	KeyTimer		: TIME := T#200ms;
	sLux_EN			: FLT_EVENT;
	chkLux_ST		: FLT_TIME := ( TTAP:=T#20S, INITEV:=FALSE );
	chkLux_ST_Analog: FLT_TIME := ( TTAP:=T#20S, INITEV:=FALSE );
	HourMinNow		: STRING;
	semaphore		: BOOL:=GRUN;
	OnFromKey		: BOOL;
	fTrigFun		: F_TRIG;
	rTrigFun		: R_TRIG;
	fTrigKey		: F_TRIG;
	ActionKeyState	: en_ActionKey;
	KeyCounter, x	: BYTE;
	CtrlKey			: BOOL;
	DimmingValForKey: INT; (* valore 0...100 del dimming di default del lux sotto key *)
	ModeToServer : BYTE;
	ForcedOn : BYTE;
	ForcedOff : BYTE;

END_VAR
(* Con l'ID si identifica il numero del lux sul campo quindi il suo valore può variare da 1 a LUXM_MAX (attualmente 1...900) *)
IF (KeyMode = BUTTON_NO) OR (KeyMode = BUTTON_NC) THEN (* se si usano dei pulsanti sui vari digital input...*)
	KeyCounter := 0;
	FOR x:=0 TO  KeyQty-1 DO
		IF CtrlKeyList[x] = 1 THEN
			KeyCounter := KeyCounter + 1;
		END_IF
	END_FOR
	IF (KeyCounter MOD 2) = 0 THEN
		CtrlKey := FALSE;
	ELSE
		DimmingValForKey := DimmingValForKeyList[0]; (* In caso di pulsanti si prende il valore della posizione 0 dell'array *)
		CtrlKey := TRUE;
	END_IF
ELSE (* altrimenti se uso l'interruttore ne posso usare solo 1 nella posizione 0 dell'array *)
	IF (DimmingValForKeyMax) THEN
		DimmingValForKey := 0;
		FOR x:=0 TO  KeyQty-1 DO
			IF (CtrlKeyList[x] = 1) AND (DimmingValForKeyList[x] > DimmingValForKey)
			THEN
				DimmingValForKey := DimmingValForKeyList[x];
			END_IF
		END_FOR
	ELSIF NOT(DimmingValForKeyMax) THEN
		DimmingValForKey :=1000;
		FOR x:=0 TO  KeyQty-1 DO
			IF (CtrlKeyList[x] = 1) AND (DimmingValForKeyList[x] < DimmingValForKey)
			THEN
				DimmingValForKey := DimmingValForKeyList[x];
			END_IF
		END_FOR
	END_IF
	CtrlKey := 0;
	FOR x:=0 TO  KeyQty-1 DO
			CtrlKey := CtrlKey OR CtrlKeyList[x];
	END_FOR

END_IF

CASE DimmingType OF (* set dell' AsiTypeOut per sapere se eseguire il set di un analog out o di un digital out *)
	NO_DIMMING:	(* if no dimming we are using a digital output *)
		LuxTypeOut := DIGITAL; (* Set digital out mode *)
	DIMMING:	(*  if dimming we are using analog output *)
		LuxTypeOut := ANALOG; (* Set analog out mode *)
END_CASE

(* Control logic *)
(* Restore mode and value	*)
IF RestoreKey THEN
	CTRL_MODE := CTRL_MODE_BackUp;
END_IF

CASE CTRL_MODE OF
	ManualeOff: (*  0 Manuale Off *)
		(* Se commutazione arrivata da key durante funzionamento in timer o cronografo *)
		IF  NOT(CtrlKey) AND (ActionKey > NormalMode) AND ( ActionKeyState = SwitchOFF)THEN
			ActionKeyState := NormalMode;
			CTRL_MODE := CTRL_MODE_BackUp;
		ELSE
			CASE DimmingType OF
				NO_DIMMING:	(* if no dimming we are using a digital output *)
					LuxDigitalOut := TRUE; (* Lux spento (digital) *)
				DIMMING:	(*  if dimming we are using analog and digital output *)
					DimmerCtrl(); (* In caso di switch off in manuale è sempre zero anche se arriva da key *)
			END_CASE
		END_IF
	ManualeOn: (*  1 Manuale On *)
		(* Se commutazione arrivata da key durante funzionamento in timer o cronografo *)
		IF  NOT(CtrlKey) AND (ActionKey > NormalMode) AND ( ActionKeyState = SwitchON) THEN
			ActionKeyState := NormalMode;
			CTRL_MODE := CTRL_MODE_BackUp;
		ELSE
			CASE DimmingType OF
				NO_DIMMING:	(* if no dimming we are using a digital output *)
					LuxDigitalOut := FALSE; (* Lux acceso (digital) *)
				DIMMING:	(*  if dimming we are using analog and digital output  *)
					IF ActionKeyState = SwitchON THEN
						DimmerCtrlKeyOn(); (* Se il manuale on è settato a causa di un key si impongono i dati del key stesso *)
					ELSE
						DimmerCtrl();
					END_IF
			END_CASE
		END_IF
	Cronografo: (*  2 Cronografo *)
		IF  (CtrlKey) AND (ActionKey > NormalMode) THEN
			CASE  ActionKey OF
				SwitchON: 	(* Corrisponde al manuale ON *)
					CTRL_MODE := ManualeOn;
					ActionKeyState := SwitchON;
					CASE DimmingType OF
						NO_DIMMING:	(* if no dimming we are using a digital output *)
							LuxDigitalOut := FALSE; (* Lux acceso (digital) *)
						DIMMING:	(*  if dimming we are using analog and digital output  *)
							DimmerCtrlKeyOn();
					END_CASE

				SwitchOFF:	(* Corrisponde al manuale OFF  *)
					CTRL_MODE := ManualeOff;
					ActionKeyState := SwitchOFF;
					CASE DimmingType OF
						NO_DIMMING:	(* if no dimming we are using a digital output  *)
							LuxDigitalOut := TRUE; (* Lux spento (digital)  *)
						DIMMING:	(*  if dimming we are using analog and digital output  *)
							DimmerCtrlKeyOff();
					END_CASE
			END_CASE
		ELSE
			CASE DimmingType OF
				NO_DIMMING:	(* if no dimming we are using a digital output  *)
					IF ValInCronoInLux = 1000 (* OR ( LuxElement[i].PressKeyVisuOn)  *)
						THEN
						LuxDigitalOut := FALSE; (* Lux acceso (digital)  *)
						ELSE IF ValInCronoInLux = 0 (* OR ( NOT LuxElement[i].PressKeyVisuOn)  *)
							THEN
							LuxDigitalOut := TRUE; (* Lux spento (digital)  *)
						END_IF
					END_IF
				DIMMING:	(*  if dimming we are using analog output  *)
					DimmerCtrl();
			END_CASE
		END_IF
	Timer: (*  3 Timer   *)
	IF  (CtrlKey) AND (ActionKey > NormalMode) THEN
		CASE  ActionKey OF
			SwitchON: 	(* Corrisponde al manuale ON  *)
				CTRL_MODE := ManualeOn;
				ActionKeyState := SwitchON;
				CASE DimmingType OF
					NO_DIMMING:	(* if no dimming we are using a digital output  *)
						LuxDigitalOut := FALSE; (* Lux acceso (digital)  *)
					DIMMING:	(*  if dimming we are using analog and digital output   *)
						DimmerCtrlKeyOn();
				END_CASE

			SwitchOFF:	(* Corrisponde al manuale OFF  *)
				CTRL_MODE := ManualeOff;
				ActionKeyState := SwitchOFF;
				CASE DimmingType OF
					NO_DIMMING:	(* if no dimming we are using a digital output  *)
						LuxDigitalOut := TRUE; (* Lux spento (digital)  *)
					DIMMING:	(*  if dimming we are using analog and digital output  *)
						DimmerCtrlKeyOff();
				END_CASE
		END_CASE
	ELSE
		CASE DimmingType OF
			NO_DIMMING:	(* if no dimming we are using a digital output  *)
				HourMinNow:=CONCAT('TOD#', BYTE_TO_STRING(Sys.Time_Hour));
				HourMinNow:=CONCAT(HourMinNow, ':');
				HourMinNow:=CONCAT(HourMinNow, BYTE_TO_STRING(Sys.Time_Min));
				HourMinNow:=CONCAT(HourMinNow,':00');

				(* Trig timer *)
				TrigTimer.PT:=LuxTimer;
				TrigTimer(IN:= CtrlTrig);

				IF (((STRING_TO_TOD(HourMinNow) > HourMinStartOn) AND (STRING_TO_TOD(HourMinNow) < HourMinEndOn))  (* Se siamo nell'orario corretto  *)
				OR ((LuxDigitalOut = FALSE) AND (TrigTimer.Q = FALSE))) (* oppure si era acceso e adesso siamo passati fuori orario e dobbiamo spegnere  *)
				THEN
					IF TrigTimer.Q THEN
						LuxDigitalOut := FALSE; (* Lux acceso (digital)  *)
						ELSE
							LuxDigitalOut:= TRUE; (* Lux spento (digital)  *)
					END_IF
				END_IF
			DIMMING:	(*  if dimming we are using analog output  *)

				HourMinNow:=CONCAT('TOD#', BYTE_TO_STRING(Sys.Time_Hour));
				HourMinNow:=CONCAT(HourMinNow, ':');
				HourMinNow:=CONCAT(HourMinNow, BYTE_TO_STRING(Sys.Time_Min));
				HourMinNow:=CONCAT(HourMinNow,':00');

				(* Trig timer *)
				TrigTimer.PT:=LuxTimer;
				TrigTimer(IN:= CtrlTrig);

				IF (((STRING_TO_TOD(HourMinNow) > HourMinStartOn) AND (STRING_TO_TOD(HourMinNow) < HourMinEndOn))  (* Se siamo nell'orario corretto  *)
				OR ((LuxDigitalOut = FALSE) AND (TrigTimer.Q = FALSE))) (* oppure si era acceso e adesso siamo passati fuori orario e dobbiamo spegnere  *)
				THEN
					IF TrigTimer.Q THEN
						DimmerCtrl(); (* Lux acceso  *)
						ELSE
							LuxAnalogOut := 0; (* Lux spento  *)
							LuxDigitalOut := TRUE; (* Lux spento (digital)  *)
					END_IF
				END_IF
		END_CASE
		END_IF
	KeyControl: (*  4 Key function  *)
		IF CtrlKey THEN
			CASE DimmingType OF
				NO_DIMMING:	(* if no dimming we are using a digital output  *)
					LuxDigitalOut := FALSE; (* Lux acceso (digital)  *)
				DIMMING:	(*  if dimming we are using analog and digital output   *)
					DimmerCtrlKeyOn();
			END_CASE
		ELSIF CtrlKey = 0 THEN
			CASE DimmingType OF
				NO_DIMMING:	(* if no dimming we are using a digital output  *)
					LuxDigitalOut := TRUE; (* Lux spento (digital)  *)
				DIMMING:	(*  if dimming we are using analog and digital output  *)
					DimmerCtrlKeyOff();
			END_CASE
		END_IF
	END_CASE

(* ----------------------------------------------------------------------------------------------------------------------------------------  *)
(* Se i pin del feedback relè non sono cavallottati si usa la seguente riga al posto di quelle successive indicate da(#)  *)
(* REL_ST := LUX_ST[ID];	  																					 *)
(* ----------------------------------------------------------------------------------------------------------------------------------------   *)

(* setting della variabile REL_EN per compatibilità con il sw preesistente  *)
CASE DimmingType OF
	NO_DIMMING:	(* if no dimming we are using a digital output  *)
	IF LuxDigitalOut = TRUE  (* Lux spento  *)
		THEN
			(* Lux_State := FALSE;	//A causa del cavallotto sui pin del relè forzo a falso (#)  *)
			(* Lux_State := LUX_ST[ID];	  *)
			Lux_Enable := FALSE;
		ELSIF LuxDigitalOut = FALSE  (* Lux acceso			   *)
			THEN
				(* Lux_State := LUX_ST[ID];	//Quando so che la luce è accesa leggo lo stato del pin (che essendo cavallottato sarà a 1) (#)  *)
				Lux_Enable := TRUE;
	END_IF

	DIMMING:	(*  if dimming we are using analog output  *)
	IF LuxAnalogOut  = 0 (* Lux spento				  *)
		THEN
			(* REL_ST := FALSE;	 A causa del cavallotto sui pin del relè forzo a falso (#)  *)
			(* Lux_State := LUX_ST[ID];	  *)
			Lux_State:= TRUE;	(* aggiunta perchè non ho feedback sul relè *)
			Lux_Enable := FALSE;
			Lux_EnableAnalog := LuxAnalogOut; (* GIURE ver 008   *)
		ELSIF LuxAnalogOut > 0  (* Lux acceso			  *)
			THEN
				(* Lux_State := LUX_ST[ID];	 Quando so che la luce è accesa leggo lo stato del pin (che essendo cavallottato sarà a 1) (#)  *)
				Lux_State:= TRUE; (* aggiunta perchè non ho feedback sul relè *)
				Lux_Enable := TRUE;
				Lux_EnableAnalog := LuxAnalogOut;  (* GIURE ver 008  *)
	END_IF

END_CASE
(* Temporary energy counter *)
TickTimer(IN:=NOT TickTimer.Q);
IF TickTimer.Q AND Lux_Enable THEN
	LocalWorkingTime:=LocalWorkingTime+1;
	IF LocalEnergyCounter_t>36000000 THEN
		LocalEnergyCounter_t:=LocalEnergyCounter_t-36000000;
		LocalEnergyCounter:=LocalEnergyCounter+1;
	END_IF
END_IF

(* Generate status events *)
sLux_EN(IN:=Lux_Enable);
IF sLux_EN.EVL THEN
	LogEv(EL_Log,EO_LUX,ID,2,'Light OFF'); (* Light OFF  *)
END_IF
IF sLux_EN.EVH THEN
	LogEv(EL_Log,EO_LUX,ID,3,'Light ON'); (* Light ON  *)
	LocalPowerOnCycles:=LocalPowerOnCycles+1;
END_IF


(* Check status feedback *) (* GIURE ver 008 - aggiunta controllo valori analogici  *)
chkLux_ST_Analog(IN:=(Lux_StateAnalog<>Lux_EnableAnalog));
IF chkLux_ST_Analog.EVH THEN
	LogEv(EL_Alarm,EO_LUX,ID,9,'Fail Analog');(*  Feedback failure - Lux_StateAnalog<>Lux_EnableAnalog*)
END_IF
IF chkLux_ST_Analog.EVL THEN
	LogEv(EL_Log,EO_LUX,ID,1,'Successful Analog'); (*  Light feedback OK - Lux_StateAnalog = Lux_EnableAnalog  *)
END_IF
(* Check status feedback *)
chkLux_ST(IN:=(Lux_State<>Lux_Enable));
IF chkLux_ST.EVH THEN
	LogEv(EL_Alarm,EO_LUX,ID,9,'Fail'); (*  Feedback failure - Lux_State<>Lux_Enable  *)
END_IF
IF chkLux_ST.EVL THEN
	LogEv(EL_Log,EO_LUX,ID,1,'Successful'); (*  Light feedback OK - Lux_State = Lux_Enable  *)
END_IF


(* Status color *)
IF chkLux_ST.OUT THEN
	Status_Log:=2; Status_Vis:=COLOR_RED;
ELSE
	Status_Log:=0;
	Status_Vis:=SEL(Lux_Enable,COLOR_GREEN_OFF,COLOR_GREEN);
END_IF

(* Salvataggio dati in array ordinato per numero di ID utile per la visualizzazione  *)
DataLuxForVis[ID].VisStatus:=Status_Vis;
DataLuxForVis[ID].VisTimer:=LuxTimer/1000;
DataLuxForVis[ID].VisMod:=CTRL_MODE;
(* DataLuxForVis[ID].VisMod:=any_num_to_byte(CTRL_MODE); *)
END_FUNCTION_BLOCK
ACTION AddLogData:
Logger.s1:=INSERT('&LUX=',WORD_TO_STRING(ID),4);
IF ID<10 THEN Logger.s1:=INSERT(Logger.s1,'0',4); END_IF

Logger.s1:=CONCAT(Logger.s1,BOOL_TO_STRING(Lux_Enable));				Logger.s1:=CONCAT(Logger.s1,';');
Logger.s1:=CONCAT(Logger.s1,DWORD_TO_STRING(LocalWorkingTime));		Logger.s1:=CONCAT(Logger.s1,';');
Logger.s1:=CONCAT(Logger.s1,DWORD_TO_STRING(LocalPowerOnCycles));	Logger.s1:=CONCAT(Logger.s1,';');

CASE CTRL_MODE OF		(* modifica GIURE 009 ver 1.3 *)
	0: 	(*  Manuale OFF *)
		ModeToServer := 0;
		ForcedOn := 0;
		ForcedOff := 1;
	1:	(*  Manuale ON *)
		ModeToServer := 1;
		ForcedOn := 1;
		ForcedOff := 0;
	2:	(*  Cronografo *)
		ModeToServer := 2;
		ForcedOn := 0;
		ForcedOff := 0;
	3: 	(* Timer *)
		ModeToServer := 3;
		ForcedOn := 0;
		ForcedOff := 0;
END_CASE
Logger.s1:=CONCAT(Logger.s1,BYTE_TO_STRING(ModeToServer));			Logger.s1:=CONCAT(Logger.s1,';');
Logger.s1:=CONCAT(Logger.s1,BYTE_TO_STRING(Status_Log));				Logger.s1:=CONCAT(Logger.s1,';');
Logger.s1:=CONCAT(Logger.s1,BYTE_TO_STRING(ForcedOn));				Logger.s1:=CONCAT(Logger.s1,';');
Logger.s1:=CONCAT(Logger.s1,BYTE_TO_STRING(ForcedOff));				Logger.s1:=CONCAT(Logger.s1,';');
Logger.s1:=CONCAT(Logger.s1,BYTE_TO_STRING(DimmingType));			Logger.s1:=CONCAT(Logger.s1,';');
Logger.s1:=CONCAT(Logger.s1,WORD_TO_STRING(Lux_EnableAnalog/100));

ADDSTRING(ADR(Logger.TData), ADR(Logger.s1), Logger.TLen);
END_ACTION
ACTION DimmerCtrl:
CASE CTRL_MODE OF
	0: (* Manuale Off *)
		LuxAnalogOut := 0; (* Lux spento *)
		LuxDigitalOut := TRUE; (* Lux spento (digital) *)
	1: (* Manuale On *)
		LuxAnalogOut := 10000; (* Lux acceso *)
		LuxDigitalOut := FALSE; (* Lux acceso (digital) *)
	2: (* Cronografo *)
		IF ValInCronoInLux > 0 THEN
			LuxDigitalOut := FALSE; (* Lux acceso (digital) *)
			ELSE
				LuxDigitalOut := TRUE; (* Lux spento (digital) *)
		END_IF
		LuxAnalogOut := INT_TO_WORD(ValInCronoInLux*10);
	3: (* Timer 		 *)
		IF DimmingValForTimer > 0 THEN
			LuxDigitalOut := FALSE; (* Lux acceso (digital) *)
			ELSE
				LuxDigitalOut := TRUE; (* Lux spento (digital) *)
		END_IF
		LuxAnalogOut := INT_TO_WORD(DimmingValForTimer*10);
	ELSE (* default *)
		LuxDigitalOut := FALSE; (* Lux acceso (digital) *)
		LuxAnalogOut := 10000;
END_CASE
END_ACTION
ACTION DimmerCtrlKeyOff:
LuxAnalogOut := 0; (*/Lux spento*)
LuxDigitalOut := TRUE; (*Lux spento (digital)*)
END_ACTION
ACTION DimmerCtrlKeyOn:
LuxAnalogOut := INT_TO_WORD(DimmingValForKey*10);
LuxDigitalOut := FALSE; (*Lux acceso (digital) *)
END_ACTION
ACTION StatReset:
(* Reset statistic counters *)
LocalWorkingTime:=0;
LocalPowerOnCycles:=0;
LocalEnergyCounter:=0;
END_ACTION

(* POU Plant_Objects/obj_TPV, ST *)
FUNCTION_BLOCK obj_TPV
(* === TEMPERATURE PROBE  ===
   v1.0[16/04/15] - Versioning
*)
VAR CONSTANT
	NormalEv		: BYTE := 0;
	ErrorEv			: BYTE := 1;
	WarningEv		: BYTE := 2;
END_VAR
VAR_INPUT
	(* Settings *)
	ID				: BYTE;
	TAP				: BYTE:=4;	   (* Consecutive checks filter *)
	INITEV			: BOOL:= TRUE; (* Generate init OK event *)
	IN_EMIN			: INT :=-2000; (* Low error limit *)
	IN_WMIN			: INT := -550; (* Low warning value *)
	IN_WMAX			: INT :=  900; (* High warning value *)
	IN_EMAX			: INT := 8500; (* High error limit *)
	ERR_MIN_SHORT	: BOOL:= TRUE; (* TRUE  ==> EMIN=Short        , EMAX=Disconnected
									  FALSE ==> EMIN=Disconnected , EMAX=Short 		 *)
	(* Physical input *)
	IN			: INT;
END_VAR
VAR_OUTPUT
	WRN			: BOOL;	(* Value in warning range *)
	ERR			: BOOL;	(* Value error *)
	HI			: INT;	(* Highest value - cleared by Stat_Reset() action *)
	AVG			: INT; 	(* Average value - updated by Mean() action, cleared by Mean_Reset() action *)
	LOW			: INT;	(* Lowest value  - cleared by Stat_Reset() action *)

	Status_Log	: WORD;
	Status_Vis	: DWORD;
END_VAR
VAR
	cnt			: BYTE;
	event		: BYTE := 0;	(* 0: monitoring a generic, 1: monitoring an error, 2: monitoring a warning *)
	asum		: DINT;
	acnt		: WORD;
END_VAR
(* Check probe value limits *)
IF IN<=IN_EMIN OR IN>=IN_EMAX THEN
	IF NOT ERR THEN
		IF event <> ErrorEv THEN
			cnt := 1;
			event := ErrorEv;
		ELSE
			cnt:=cnt+1;
		END_IF

		IF cnt>TAP THEN
			cnt:=0;
			ERR:=TRUE; WRN:=FALSE;
			IF ( ERR_MIN_SHORT=TRUE  AND IN<=IN_EMIN ) OR ( ERR_MIN_SHORT=FALSE AND IN>=IN_EMAX ) THEN
				LogEv(EL_Alarm,EO_TPV,ID,5,INT_TO_STRING(IN));
			ELSE
				LogEv(EL_Alarm,EO_TPV,ID,4,INT_TO_STRING(IN));
			END_IF
		END_IF
	END_IF
ELSIF IN<=IN_WMIN OR IN>=IN_WMAX THEN
	IF NOT WRN THEN
		IF event <> WarningEv THEN
			cnt := 1;
			event := WarningEv;
		ELSE
			cnt:=cnt+1;
		END_IF

		IF cnt>TAP THEN
			cnt:=0;
			ERR:=FALSE; WRN:=TRUE;
			LogEv(EL_Wrn,EO_TPV,ID,SEL(IN<=IN_WMIN,3,2),INT_TO_STRING(IN));
		END_IF
	END_IF
ELSE
	IF INITEV OR WRN OR ERR THEN
		IF event <> NormalEv THEN
			cnt := 1;
			event := NormalEv;
		ELSE
			cnt:=cnt+1;
		END_IF

		IF cnt>TAP THEN
			cnt:=0;
			INITEV:=FALSE; ERR:=FALSE; WRN:=FALSE;
			LogEv(EL_Log,EO_TPV,ID,1,'Probe_OK');
		END_IF
	END_IF
END_IF


(*
(* Average value *)
IF acnt>=500 THEN
	Mean();
	asum := asum - AVG;
	acnt := acnt - 1;
END_IF

asum := asum + IN;
acnt := acnt + 1;
*)

AVG := IN;



(* Statistics values *)
IF IN<LOW THEN LOW:=IN; END_IF
IF IN>HI  THEN HI :=IN; END_IF

Lamp.obj_Status := Status_Log;
Lamp.UpdateStatus();

(* Status Log *)
IF ERR THEN	Status_Log := 2; Status_Vis := COLOR_RED;
ELSIF WRN THEN Status_Log := 1;	Status_Vis := COLOR_YELLOW;
ELSE Status_Log := 0; Status_Vis := COLOR_GREEN;
END_IF
END_FUNCTION_BLOCK
ACTION AddLogData:
Logger.s1:=INSERT('&TPV=',BYTE_TO_STRING(ID),4);
IF ID<10 THEN Logger.s1:=INSERT(Logger.s1,'0',4); END_IF
(*
Mean();
*)
Logger.s1:=CONCAT(Logger.s1,INT_TO_STRING(AVG));		Logger.s1:=CONCAT(Logger.s1,';');

Logger.s1:=CONCAT(Logger.s1,WORD_TO_STRING(Status_Log));
ADDSTRING(ADR(Logger.TData), ADR(Logger.s1), Logger.TLen);
END_ACTION
ACTION Mean:
(*AVG := DINT_TO_INT(asum/acnt); *)


AVG := IN;
END_ACTION
ACTION Mean_Reset:
AVG:=IN;
asum:=IN;
acnt:=1;
END_ACTION
ACTION Stat_Reset:
HI:=IN;
LOW:=IN;
END_ACTION

(* POU Plant_Objects/obj_VRD_new, ST *)
FUNCTION_BLOCK obj_VRD_new
(* === VALVOLA RIPARTITORE ===
   v1.0[16/04/15] - Versioning
*)
VAR CONSTANT
	Chk_CntSecAlarm	: INT := 900;	(* 900s = 15 minutes -> Observation itme *)
END_VAR
VAR_INPUT
	(* Settings *)
	ID				: BYTE;
	(* Controls *)
	RUN  			: BOOL;					(* Control input *)
	ReducedRange	: BOOL := FALSE;		(* If true output value is among 2 and 10V, otherwise 0-10V *)

	(* Physical inputs *)
	TEMP 			: INT;		(* Input temperature from sensor *)
	STATUS 			: WORD;		(* Input position from valve *)

	InitOK			: BOOL;
	Alarm1			: BOOL;
	Alarm2			: BOOL;
	Warning			: BOOL;

	Ctrl_Init		: BOOL;
	Ctrl_SetPoint	: INT;
	Ctrl_SetPointNew: INT := 0;
	Delta_SetPoint	: INT;
	Ctrl_Err		: INT;			(* Current error *)
	Ctrl_Err0		: INT; 			(* Previous error *)
	Ctrl_Accel		: REAL;			(* Derivate of error *)
	Ctrl_AccelGate  : INT:=1;		(* Derivate gate *)
	Ctrl_AccelTmr	: WORD;
	Ctrl_SetPointGate: INT := 5;	(* Setpoint gate - 0.5°C *)
	Ctrl_ErrGate	: INT:=5;		(* Error gate *)
	Ctrl_Kp			: REAL:=2;(*1;*)		(* Proportional factor *)
	Ctrl_Kd			: REAL:=10;(*100;*)  	(* Derivative factor *)
	Ctrl_Out		: REAL;

	Chk_Err			: INT;
	Chk_ErrGate		: INT:=1000; 		(* Check error gate *)
	Chk_Cnt			: INT;
	Chk_CntAlarm	: INT:=240; 		(* Check error trigger 120s *)

	(* Status *)
	Log_AvgTemp		: AVERAGE_T;
	Status_Log		: BYTE;
	Status_Vis 		: DWORD;

	(* Feedback *)
	fFeedback		: BOOL;			(* TRUE: Feedback available, FALSE: Feedback not available *)

	OffsetBoost: INT;

END_VAR
VAR_IN_OUT
(*	CLIM		: typ_Clima;  *)
END_VAR
VAR_OUTPUT
	(* Physical outputs *)
	OUT			: WORD;
END_VAR
VAR
	Curve		: CHARCURVE;
	Curve_Err	: BYTE;

	aTemp		: ARRAY [1..20] OF INT;
	meanTemp	: INT;
	sum			: INT := 0;
	Tmr			: TON := (PT:=T#1s);
	index		: BYTE;
	i			: BYTE;
	fCtrl_Err	: BOOL;		(* TRUE: Ctrl_Err>0, FALSE: Ctrl_Err<0 *)

	TON_AllarmeOvertemperatura:TON;


END_VAR


VAR_INPUT RETAIN
	Local_VRD_TAlarm: INT;
END_VAR
(* Check initialization *)
(*IF NOT InitOK THEN Init(); END_IF*)

(* Check max temperature *)

TON_AllarmeOvertemperatura(IN:=TEMP>Local_VRD_TAlarm,PT:=t#20s);
IF TON_AllarmeOvertemperatura.Q THEN
	IF NOT Alarm1 THEN
		Alarm1:=TRUE;
		LogEv(EL_AlarmStop,EO_VRD,ID,3,'VRD_Overtemperature');
	END_IF
END_IF

IF (TEMP<Local_VRD_TAlarm-10) AND Alarm1  THEN
		Alarm1:=FALSE;
END_IF




(* Check climatic setup *)
IF NOT CLIM.InitOK THEN	DefaultClim(); END_IF;
(* Calculate Setpoint *)
Curve(	IN:= T_AMB,	N:= 5, P:= CLIM.Points,			(* Given the x value as input, the corresponding y value as output is returned, if it matches the crve designed by array of points *)
		OUT=> Ctrl_SetPointNew, ERR=> Curve_Err );

IF Curve_Err>0 OR Ctrl_SetPoint>Plant_VRD_TMax THEN
	Ctrl_SetPoint:=Plant_VRD_TDefault;
	IF NOT Warning THEN
		Warning:=TRUE;
		LogEv(EL_Wrn,EO_VRD,ID,2,'VRD_Climatic_Error');
	END_IF
ELSE
	Delta_SetPoint := ABS(Ctrl_SetPoint - Ctrl_SetPointNew);
	IF Delta_SetPoint>Ctrl_SetPointGate THEN Ctrl_SetPoint := Ctrl_SetPointNew; END_IF

	Warning:=FALSE;
END_IF

Ctrl_SetPoint:=Ctrl_SetPoint+OffsetBoost;


(* Execute control loop [T=500ms] *)
(* IF RUN AND (NOT Alarm1) THEN*)
IF RUN  THEN
	(* Calculate error *)
	Ctrl_Err:=Ctrl_SetPoint-TEMP;
	(* Init/restart operations *)
	IF NOT Ctrl_Init THEN
		Ctrl_Accel:=0;
		Ctrl_AccelTmr:=0;
		Ctrl_Err0:=Ctrl_Err;
		Ctrl_Out:=5000;
		Ctrl_Init:=TRUE;
	END_IF
	(* Calculate acceleration *)
	IF ABS(Ctrl_Err-Ctrl_Err0)>Ctrl_AccelGate OR Ctrl_AccelTmr>20 THEN
		Ctrl_Accel:=INT_TO_REAL(Ctrl_Err-Ctrl_Err0)/WORD_TO_REAL(1+Ctrl_AccelTmr);
		Ctrl_AccelTmr:=0;
		Ctrl_Err0:=Ctrl_Err;
	ELSE
		Ctrl_AccelTmr:=Ctrl_AccelTmr+1;
	END_IF

	(* Gate error *)
	IF ABS(Ctrl_Err)>Ctrl_ErrGate THEN
		(* Control loop *)
		Ctrl_Out:=Ctrl_Out+(Ctrl_Kp*Ctrl_Err)+(Ctrl_Kd*Ctrl_Accel);
	END_IF

	(* Limiter and Output *)
(*	Ctrl_Out:=LIMIT(0,Ctrl_Out,27000); *)
	Ctrl_Out:=LIMIT(0,Ctrl_Out,32000);

ELSE
	Ctrl_Init:=FALSE;
	Ctrl_Out:=0;
END_IF

OUT:=SEL(Alarm1,REAL_TO_WORD(Ctrl_Out),0);





(* If there is an hardware feedback (such as 0-10V, potentiometer, ...) check it otherwise try to rebuild it *)
IF fFeedback THEN CheckFeedback();
ELSE BuildFeedback();
END_IF

(* Status temp *)
(* Status color *)
   IF Alarm1 THEN Status_Log:=2; Status_Vis:=16#2020F0;
ELSIF Warning  OR Alarm2        THEN Status_Log:=1; Status_Vis:=16#20F0F0;
                       ELSE Status_Log:=0; Status_Vis:=SEL(RUN,16#006000,16#20F020);
END_IF
END_FUNCTION_BLOCK
ACTION AddLogData:
Logger.s1:=INSERT('&VRD=',BYTE_TO_STRING(ID),4);
IF ID<10 THEN Logger.s1:=INSERT(Logger.s1,'0',4); END_IF


Logger.s1:=CONCAT(Logger.s1,INT_TO_STRING(Ctrl_SetPoint));				Logger.s1:=CONCAT(Logger.s1,';');

(* gli passo la percentuale di comando che ricavo dalla divisone per 327 del comando fisico *)
Logger.s1:=CONCAT(Logger.s1,WORD_TO_STRING(OUT/327));						Logger.s1:=CONCAT(Logger.s1,';');


(* gli passo la percentuale di apertura che ricavo dalla divisone per 327 del comando fisico *)
IF fFeedback THEN Logger.s1:=CONCAT(Logger.s1,WORD_TO_STRING(STATUS/327));
ELSE Logger.s1:=CONCAT(Logger.s1,'0');	(* Bypass *)
END_IF

Logger.s1:=CONCAT(Logger.s1,';');

Logger.s1:=CONCAT(Logger.s1,WORD_TO_STRING(Status_Log));

Logger.s1:=CONCAT(Logger.s1,';');
Logger.s1:=CONCAT(Logger.s1,'1'); (* Valvola modulante controllata Analogica *)

ADDSTRING(ADR(Logger.TData), ADR(Logger.s1), Logger.TLen);
END_ACTION
ACTION BuildFeedback:
(* Comparison is taken between actual temperature vs windowed mean value of last 20 temperature
   (check is carried out every second)	*)
IF RUN AND (NOT Alarm1) THEN

	IF Ctrl_Err>0 THEN
		IF NOT fCtrl_Err THEN index := 0; END_IF
		fCtrl_Err := TRUE;
	ELSE
		IF fCtrl_Err THEN index := 0; END_IF
		fCtrl_Err := FALSE;
	END_IF

	(* Temperature is lower than setpoint -->> Should increase *)
	Tmr(IN:=NOT Tmr.Q);

	IF Tmr.Q THEN

		IF index<21 THEN
			(* Fullfil temperature array *)
			aTemp[index] := TEMP;
			index := index + 1;

			IF index=20 THEN
				FOR i:=1 TO 20 BY 1 DO sum := sum + aTemp[i]; END_FOR
			END_IF
		ELSE
			(* Calculate mean value *)
			meanTemp := sum/20;

			IF (fCtrl_Err AND TEMP<meanTemp) OR (NOT fCtrl_Err AND TEMP>meanTemp) THEN

				IF Chk_Cnt>Chk_CntSecAlarm THEN
					IF NOT Alarm2 THEN
						Alarm2:=TRUE;
						LogEv(EL_Alarm,EO_VRD,ID,4,'VRD_Position_Error');
					END_IF
				ELSE
					Chk_Cnt := Chk_Cnt+1;
				END_IF

			ELSE
				(* Reset counter and alarm flag *)
				Chk_Cnt:=0;
				Alarm2:=FALSE;
			END_IF

			sum := 0;	(* Reset sum counter *)

			(* Shift array removing oldest value *)
			FOR i:=1 TO 20 BY 1 DO
				aTemp[i-1] := aTemp[i];
				sum := sum + aTemp[i];
			END_FOR

			aTemp[20] := TEMP;			(* Last temperature value is new one *)
			sum := sum + aTemp[20];		(* Update sum *)
		END_IF
	END_IF
END_IF
END_ACTION
ACTION CheckFeedback:
(* Calculate position error according to feedback *)
IF ReducedRange THEN
(* SETPOINT[2..10V]-STATUS[0..10V] *)
	IF OUT<=6553 THEN Chk_Err:=0; ELSE Chk_Err:=(OUT-6553)/262; END_IF
	Chk_Err:=(Chk_Err-STATUS)/327;
ELSE
(* SETPOINT[0..10V]-STATUS[0..10V] *)
	Chk_Err := OUT - STATUS;
END_IF

(* Check position error *)
IF ( ABS(Chk_Err)>Chk_ErrGate ) THEN
	IF Chk_Cnt>Chk_CntAlarm THEN
		IF NOT Alarm2 THEN
			Alarm2:=TRUE;
			LogEv(EL_Wrn,EO_VRD,ID,4,'VRD_Position_Error');
		END_IF
	ELSE
		Chk_Cnt:=Chk_Cnt+1;
	END_IF
ELSE
	Chk_Cnt:=0;
	Alarm2:=FALSE;
END_IF
END_ACTION
ACTION DefaultClim:
(*CLIM.Points[0].X:=-300; CLIM.Points[0].Y:=400;
CLIM.Points[1].X:=-50;  CLIM.Points[1].Y:=400;
CLIM.Points[2].X:= 200; CLIM.Points[2].Y:=200;
CLIM.Points[3].X:= 300; CLIM.Points[3].Y:=200;
CLIM.Points[4].X:= 500; CLIM.Points[4].Y:=200;*)
CLIM.Points[0].X:=-300; CLIM.Points[0].Y:=850;
CLIM.Points[1].X:=-50;  CLIM.Points[1].Y:=650;
CLIM.Points[2].X:= 100; CLIM.Points[2].Y:=400;
CLIM.Points[3].X:= 200; CLIM.Points[3].Y:=200;
CLIM.Points[4].X:= 500; CLIM.Points[4].Y:=200;
CLIM.InitOK:=TRUE;
LogEv(EL_Wrn,EO_VRD,ID,1,'Climatic_Default');
END_ACTION
ACTION Init:
(* End initialization *)
InitOK:=TRUE;
END_ACTION

(* POU Utils Functions/PLANT_STATUS, ST *)
FUNCTION_BLOCK PLANT_STATUS
VAR_INPUT
	obj_Status		:	WORD;
END_VAR
VAR_OUTPUT
END_VAR
VAR
	PLANT_STATUS	:	WORD;

	Pwm				:	TON := (PT:=T#1s);
END_VAR
CASE plant_Status OF

	0:	(* Plant OK - Everything works well *)
		(*Pwm(IN:=FALSE);	*)						(* Stop timer if running *)
		LAMP_AL := FALSE;						(* Keep the lamp switched off *)

	(*1:	(* Plant in warning *)
		Pwm(IN:= NOT(Pwm.Q));

		IF Pwm.Q THEN
			LAMP_AL := NOT LAMP_AL;				(* Toggle output *)
		END_IF*)

	2:	(* Plant in alarm *)
		(*Pwm(IN:=FALSE);	*)						(* Stop timer if running *)
		LAMP_AL	:= TRUE;						(* Keep the lamp switched on *)

END_CASE

plant_Status := 0;		(* Reset plant status *)
END_FUNCTION_BLOCK
ACTION UpdateStatus:
IF plant_Status = 2 THEN

	RETURN;					(* If plant already in alarm condition do nothing *)

ELSE

		IF obj_Status <> 0 THEN
			plant_Status := obj_Status;			(* If plant in warning/normal condition and current object in alarm, update plant status *)
		END_IF
END_IF
END_ACTION

(* POU PLC_WDT, ST *)
FUNCTION PLC_WDT: DWORD VAR_INPUT dwEvent: DWORD; dwFilter: DWORD; dwOwner: DWORD; END_VAR
LogEv(EL_AlarmStop,EO_SYS,1,10,'Watchdog');
END_FUNCTION

(* POU Utils Functions/RAWTOHEXSTR, ST *)
FUNCTION RAWTOHEXSTR : STRING(128)
VAR_INPUT
	pData: POINTER TO BYTE;
	DataLen: BYTE;
END_VAR
VAR
	pt: POINTER TO BYTE;
	xl: BYTE;
END_VAR
pt:=ADR(RAWTOHEXSTR);

xl:=2;

WHILE DataLen>0 AND xl<128 DO

	pt^ := (pData^ / 16#10) + 48 + (((pData^ / 16#10)/10)*7);
	pt:=pt+1;
	pt^ := (pData^ AND 16#0F)  + 48 + (((pData^ AND 16#0F)/10)*7);
	pt:=pt+1;

	xl:=xl+2;

	DataLen:=DataLen-1;
	pData:=pData+1;

END_WHILE

pt^:=0;
END_FUNCTION

(* POU Utils/RTC_Update, ST *)
FUNCTION RTC_Update : BOOL
VAR
	T: DT;
	TS: STRING;
	TS2: STRING;
	Hour: BYTE;
	Minute: BYTE;
END_VAR
(* Get RTC time *)
T:=SysRtcGetTime(TRUE);
Sys.Time_CT_DT:=T;
(* Calculate variables *)
TS:=DT_TO_STRING(T);
Sys.Time_LogString:=DELETE(STR:=TS, LEN:=3, POS:=1);
TS2:=MID(STR:=TS, LEN:=4, POS:= 4); Sys.Time_Year 	:=STRING_TO_WORD(TS2);
TS2:=MID(STR:=TS, LEN:=2, POS:= 9); Sys.Time_Month	:=STRING_TO_BYTE(TS2);
TS2:=MID(STR:=TS, LEN:=2, POS:=12); Sys.Time_Day  	:=STRING_TO_BYTE(TS2);
Sys.Time_CT_Day:=(32*(Sys.Time_Month-1)+Sys.Time_Day-1);
TS2:=MID(STR:=TS, LEN:=2, POS:=15); Hour			:=STRING_TO_BYTE(TS2);
TS2:=MID(STR:=TS, LEN:=2, POS:=18); Minute		 	:=STRING_TO_BYTE(TS2);
Sys.Time_Hour := Hour;
Sys.Time_Minute := Minute;
Sys.Time_CT_Quarter:=Hour*4+(Minute/15);
Sys.Time_CT_Minute:=Hour*60+Minute;
END_FUNCTION

(* POU Utils Functions/SHIFT_ARRAY, ST *)
FUNCTION SHIFT_ARRAY : BOOL
VAR_INPUT
	pData	:	POINTER TO ARRAY [1..2] OF WORD;
	Size	:	BYTE;
END_VAR
VAR
	pNew	:	POINTER TO WORD;
	i		:	BYTE;
END_VAR
(* Shift right *)
FOR i:=1 TO (Size-1) BY 1 DO

	(*pNew := pData + 1;*)
	pData^[i] := pData^[i+1];
	(*pData := pData + 1;*)

END_FOR
END_FUNCTION

(* POU Utils Functions/TONOF, ST *)
FUNCTION_BLOCK TONOF
VAR_INPUT
	IN		: BOOL;
	PT_ON	: TIME; (* time to pass, before OUT is set *)
	PT_OF	: TIME; (* time to pass, before OUT is reset *)
END_VAR
VAR_OUTPUT
	OUT		: BOOL;
END_VAR
VAR
	timer	: TON;
END_VAR
IF IN<>OUT THEN
	timer(IN:=TRUE,PT:=SEL(IN,PT_OF,PT_ON));
	IF timer.Q THEN OUT:=IN; END_IF
ELSE
	timer(IN:=FALSE);
END_IF
END_FUNCTION_BLOCK

(* Visualisation PLC_VISU
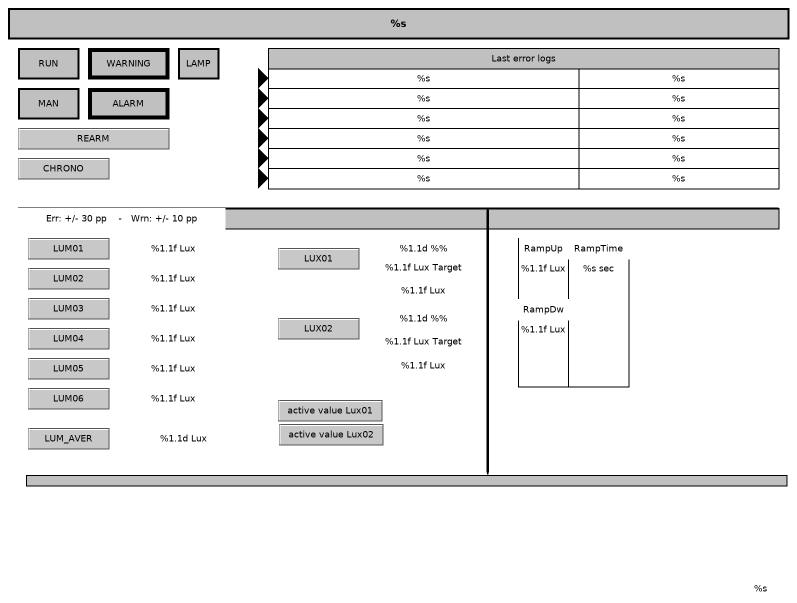
rectangle at (10,10)-(791,41): text "%s"; shows .Plant_NAME
rectangle at (530,580)-(771,601): text "%s"; shows Sys.Time_LogString
rounded rectangle at (20,50)-(81,81): text "RUN"; alarm colour if NOT Mode_Manual; runs INTERN ASSIGN Mode_Manual:=(FALSE)
rounded rectangle at (20,90)-(81,121): text "MAN"; alarm colour if Mode_Manual; runs INTERN ASSIGN Mode_Manual:=(TRUE)
rectangle at (580,70)-(781,91): text "%s"; shows Sys.LastLogs_Msg[0]
polygon at (260,170)-(270,190): invisible if Sys.LastLogs_Idx<>0
rectangle at (580,90)-(781,111): text "%s"; shows Sys.LastLogs_Msg[1]
polygon at (260,70)-(270,90): invisible if Sys.LastLogs_Idx<>1
rectangle at (580,110)-(781,131): text "%s"; shows Sys.LastLogs_Msg[2]
polygon at (260,90)-(270,110): invisible if Sys.LastLogs_Idx<>2
rectangle at (580,130)-(781,151): text "%s"; shows Sys.LastLogs_Msg[3]
polygon at (260,110)-(270,130): invisible if Sys.LastLogs_Idx<>3
rectangle at (580,150)-(781,171): text "%s"; shows Sys.LastLogs_Msg[4]
polygon at (260,130)-(270,150): invisible if Sys.LastLogs_Idx<>4
rectangle at (580,170)-(781,191): text "%s"; shows Sys.LastLogs_Msg[5]
polygon at (260,150)-(270,170): invisible if Sys.LastLogs_Idx<>5
rectangle at (270,70)-(581,91): text "%s"; shows Sys.LastLogs_Dat[0]
rectangle at (270,90)-(581,111): text "%s"; shows Sys.LastLogs_Dat[1]
rectangle at (270,110)-(581,131): text "%s"; shows Sys.LastLogs_Dat[2]
rectangle at (270,130)-(581,151): text "%s"; shows Sys.LastLogs_Dat[3]
rectangle at (270,150)-(581,171): text "%s"; shows Sys.LastLogs_Dat[4]
rectangle at (270,170)-(581,191): text "%s"; shows Sys.LastLogs_Dat[5]
rectangle at (90,90)-(171,121): text "ALARM"; alarm colour if Sys.Alarm; runs INTERN ASSIGN Mode_Manual:=(FALSE)
rectangle at (90,50)-(171,81): text "WARNING"; alarm colour if Sys.Warning; runs INTERN ASSIGN Mode_Manual:=(TRUE)
button at (20,130)-(171,151): text "REARM"; runs INTERN ASSIGN Sys.Alarm:=(FALSE);INTERN ASSIGN Sys.Warning:=(FALSE)
rectangle at (270,50)-(781,71): text "Last error logs"
rectangle at (520,240)-(571,261): text "RampUp"
rectangle at (520,260)-(571,281): text "%1.1f Lux"; shows RampUp*LuxSuBit
rounded rectangle at (180,50)-(221,81): text "LAMP"; alarm colour if LAMP_AL
button at (20,160)-(111,181): text "CHRONO"; opens VIS_CHONOEDITOR
button at (30,240)-(111,261): text "LUM01"
rectangle at (130,240)-(221,261): text "%1.1f Lux"; shows INT_TO_REAL(LumList[1].IN)*LuxSuBit
button at (30,270)-(111,291): text "LUM02"
rectangle at (130,270)-(221,291): text "%1.1f Lux"; shows INT_TO_REAL(LumList[2].IN)*LuxSuBit
button at (30,300)-(111,321): text "LUM03"
rectangle at (130,300)-(221,321): text "%1.1f Lux"; shows INT_TO_REAL(LumList[3].IN)*LuxSuBit
button at (30,330)-(111,351): text "LUM04"
rectangle at (130,330)-(221,351): text "%1.1f Lux"; shows INT_TO_REAL(LumList[4].IN)*LuxSuBit
button at (30,360)-(111,381): text "LUM05"
rectangle at (130,360)-(221,381): text "%1.1f Lux"; shows INT_TO_REAL(LumList[5].IN)*LuxSuBit
button at (30,390)-(111,411): text "LUM06"
rectangle at (130,390)-(221,411): text "%1.1f Lux"; shows DWORD_TO_REAL(LumList[6].IN)*LuxSuBit
button at (30,430)-(111,451): text "LUM_AVER"
rectangle at (140,430)-(231,451): text "%1.1d Lux"; shows PLC_PRG.LumValueAverageLux
button at (280,250)-(361,271): text "LUX01"
rectangle at (380,240)-(471,261): text "%1.1d %%"; shows LuxOutput[1].AnalogOut/100
rectangle at (380,282)-(471,303): text "%1.1f Lux"; shows INT_TO_REAL(LUX01)*LuxSuBit
button at (280,320)-(361,341): text "LUX02"
rectangle at (380,310)-(471,331): text "%1.1d %%"; shows LuxOutput[2].AnalogOut/100
rectangle at (380,357)-(471,378): text "%1.1f Lux"; shows INT_TO_REAL(LUX02)*LuxSuBit
rectangle at (520,301)-(571,322): text "RampDw"
rectangle at (520,321)-(571,342): text "%1.1f Lux"; shows RampDown*LuxSuBit
rectangle at (570,240)-(631,261): text "RampTime"
rectangle at (570,260)-(631,281): text "%s sec"; shows RampTime
rectangle at (20,210)-(227,231): text "Err: +/- 30 pp    -   Wrn: +/- 10 pp"
button at (280,402)-(384,423): text "active value Lux01"; toggles PLC_PRG.ValInCronoFromVisu[1]
button at (281,426)-(385,447): text "active value Lux02"; toggles PLC_PRG.ValInCronoFromVisu[2]
rectangle at (380,333)-(471,354): text "%1.1f Lux Target"; shows LuxOutput[2].AnalogOut*3.27*LuxSuBit
rectangle at (380,259)-(471,280): text "%1.1f Lux Target"; shows LuxOutput[1].AnalogOut*3.27*LuxSuBit
7 more shapes without text or variables
10 elements of other kinds (tables, trends, ...) not read
*)

(* Visualisation VIS_CHONOEDITOR
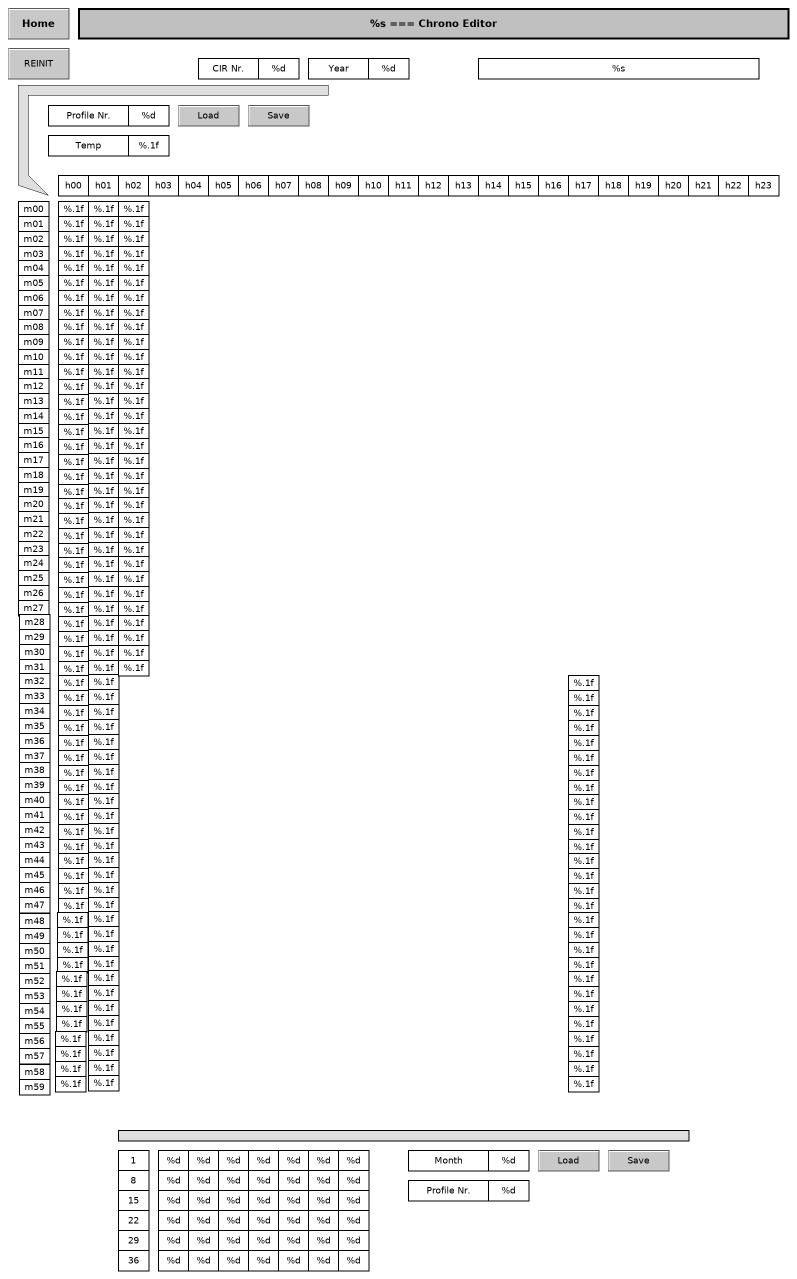
rectangle at (200,60)-(261,81): text "CIR Nr."
rectangle at (260,60)-(301,81): text "%d"; shows CronEd.CN_Sel; alarm colour if CronEd.CN_Sel<>CronEd.CN_Act; editable 1..250
rectangle at (50,107)-(131,128): text "Profile Nr."
rectangle at (130,107)-(171,128): text "%d"; shows CronEd.PR_Sel; alarm colour if CronEd.PR_Sel<>CronEd.PR_Act; editable 1..10
rectangle at (50,137)-(131,158): text "Temp"
rectangle at (130,137)-(171,158): text "%.1f"; shows CronEd.PR_TT; editable
button at (180,107)-(241,128): text "Load"; toggles CronEd.PR_Load
button at (250,107)-(311,128): text "Save"; toggles CronEd.PR_Save
rectangle at (20,203)-(51,219): text "m00"
rectangle at (20,218)-(51,234): text "m01"
rectangle at (20,233)-(51,249): text "m02"
rectangle at (20,248)-(51,264): text "m03"
rectangle at (80,10)-(791,41): text "%s === Chrono Editor"; shows .Plant_NAME
button at (10,10)-(71,41): text "Home"; opens PLC_VISU
rounded rectangle at (60,203)-(91,219): text "%.1f"; shows WORD_TO_REAL(CronEd.PR.Setpoint[0])/10; runs INTERN ASSIGN CronEd.PR.Setpoint[0]:=(REAL_TO_WORD(CronEd.PR_TT*10))
rounded rectangle at (60,218)-(91,234): text "%.1f"; shows WORD_TO_REAL(CronEd.PR.Setpoint[1])/10; runs INTERN ASSIGN CronEd.PR.Setpoint[1]:=(REAL_TO_WORD(CronEd.PR_TT*10))
rounded rectangle at (60,233)-(91,249): text "%.1f"; shows WORD_TO_REAL(CronEd.PR.Setpoint[2])/10; runs INTERN ASSIGN CronEd.PR.Setpoint[2]:=(REAL_TO_WORD(CronEd.PR_TT*10))
rounded rectangle at (60,248)-(91,264): text "%.1f"; shows WORD_TO_REAL(CronEd.PR.Setpoint[3])/10; runs INTERN ASSIGN CronEd.PR.Setpoint[3]:=(REAL_TO_WORD(CronEd.PR_TT*10))
rectangle at (60,177)-(91,198): text "h00"; runs INTERN ASSIGN CronEd.PR.Setpoint[0]:=(REAL_TO_WORD(CronEd.PR_TT*10));INTERN ASSIGN CronEd.PR.Setpoint[1]:=(REAL_TO_WORD(CronEd.PR_TT*10));INTERN ASSIGN CronEd.PR.Setpoint[2]:=(REAL_TO_WORD(CronEd.PR_TT*10));INTERN ASSIGN CronEd.PR.Setpoint[3]:=(REAL_TO_WORD(CronEd.PR_TT*10))
rectangle at (90,177)-(121,198): text "h01"; runs INTERN ASSIGN CronEd.PR.Setpoint[4]:=(REAL_TO_WORD(CronEd.PR_TT*10));INTERN ASSIGN CronEd.PR.Setpoint[5]:=(REAL_TO_WORD(CronEd.PR_TT*10));INTERN ASSIGN CronEd.PR.Setpoint[6]:=(REAL_TO_WORD(CronEd.PR_TT*10));INTERN ASSIGN CronEd.PR.Setpoint[7]:=(REAL_TO_WORD(CronEd.PR_TT*10))
rectangle at (120,177)-(151,198): text "h02"; runs INTERN ASSIGN CronEd.PR.Setpoint[8]:=(REAL_TO_WORD(CronEd.PR_TT*10));INTERN ASSIGN CronEd.PR.Setpoint[9]:=(REAL_TO_WORD(CronEd.PR_TT*10));INTERN ASSIGN CronEd.PR.Setpoint[10]:=(REAL_TO_WORD(CronEd.PR_TT*10));INTERN ASSIGN CronEd.PR.Setpoint[11]:=(REAL_TO_WORD(CronEd.PR_TT*10))
rectangle at (150,177)-(181,198): text "h03"; runs INTERN ASSIGN CronEd.PR.Setpoint[15]:=(REAL_TO_WORD(CronEd.PR_TT*10));INTERN ASSIGN CronEd.PR.Setpoint[14]:=(REAL_TO_WORD(CronEd.PR_TT*10));INTERN ASSIGN CronEd.PR.Setpoint[13]:=(REAL_TO_WORD(CronEd.PR_TT*10));INTERN ASSIGN CronEd.PR.Setpoint[12]:=(REAL_TO_WORD(CronEd.PR_TT*10))
rectangle at (180,177)-(211,198): text "h04"; runs INTERN ASSIGN CronEd.PR.Setpoint[19]:=(REAL_TO_WORD(CronEd.PR_TT*10));INTERN ASSIGN CronEd.PR.Setpoint[18]:=(REAL_TO_WORD(CronEd.PR_TT*10));INTERN ASSIGN CronEd.PR.Setpoint[17]:=(REAL_TO_WORD(CronEd.PR_TT*10));INTERN ASSIGN CronEd.PR.Setpoint[16]:=(REAL_TO_WORD(CronEd.PR_TT*10))
rectangle at (210,177)-(241,198): text "h05"; runs INTERN ASSIGN CronEd.PR.Setpoint[23]:=(REAL_TO_WORD(CronEd.PR_TT*10));INTERN ASSIGN CronEd.PR.Setpoint[22]:=(REAL_TO_WORD(CronEd.PR_TT*10));INTERN ASSIGN CronEd.PR.Setpoint[21]:=(REAL_TO_WORD(CronEd.PR_TT*10));INTERN ASSIGN CronEd.PR.Setpoint[20]:=(REAL_TO_WORD(CronEd.PR_TT*10))
rectangle at (240,177)-(271,198): text "h06"; runs INTERN ASSIGN CronEd.PR.Setpoint[27]:=(REAL_TO_WORD(CronEd.PR_TT*10));INTERN ASSIGN CronEd.PR.Setpoint[26]:=(REAL_TO_WORD(CronEd.PR_TT*10));INTERN ASSIGN CronEd.PR.Setpoint[25]:=(REAL_TO_WORD(CronEd.PR_TT*10));INTERN ASSIGN CronEd.PR.Setpoint[24]:=(REAL_TO_WORD(CronEd.PR_TT*10))
rectangle at (270,177)-(301,198): text "h07"; runs INTERN ASSIGN CronEd.PR.Setpoint[31]:=(REAL_TO_WORD(CronEd.PR_TT*10));INTERN ASSIGN CronEd.PR.Setpoint[30]:=(REAL_TO_WORD(CronEd.PR_TT*10));INTERN ASSIGN CronEd.PR.Setpoint[29]:=(REAL_TO_WORD(CronEd.PR_TT*10));INTERN ASSIGN CronEd.PR.Setpoint[28]:=(REAL_TO_WORD(CronEd.PR_TT*10))
rectangle at (300,177)-(331,198): text "h08"; runs INTERN ASSIGN CronEd.PR.Setpoint[35]:=(REAL_TO_WORD(CronEd.PR_TT*10));INTERN ASSIGN CronEd.PR.Setpoint[34]:=(REAL_TO_WORD(CronEd.PR_TT*10));INTERN ASSIGN CronEd.PR.Setpoint[33]:=(REAL_TO_WORD(CronEd.PR_TT*10));INTERN ASSIGN CronEd.PR.Setpoint[32]:=(REAL_TO_WORD(CronEd.PR_TT*10))
rectangle at (330,177)-(361,198): text "h09"; runs INTERN ASSIGN CronEd.PR.Setpoint[39]:=(REAL_TO_WORD(CronEd.PR_TT*10));INTERN ASSIGN CronEd.PR.Setpoint[38]:=(REAL_TO_WORD(CronEd.PR_TT*10));INTERN ASSIGN CronEd.PR.Setpoint[37]:=(REAL_TO_WORD(CronEd.PR_TT*10));INTERN ASSIGN CronEd.PR.Setpoint[36]:=(REAL_TO_WORD(CronEd.PR_TT*10))
rectangle at (360,177)-(391,198): text "h10"; runs INTERN ASSIGN CronEd.PR.Setpoint[43]:=(REAL_TO_WORD(CronEd.PR_TT*10));INTERN ASSIGN CronEd.PR.Setpoint[42]:=(REAL_TO_WORD(CronEd.PR_TT*10));INTERN ASSIGN CronEd.PR.Setpoint[41]:=(REAL_TO_WORD(CronEd.PR_TT*10));INTERN ASSIGN CronEd.PR.Setpoint[40]:=(REAL_TO_WORD(CronEd.PR_TT*10))
rectangle at (390,177)-(421,198): text "h11"; runs INTERN ASSIGN CronEd.PR.Setpoint[47]:=(REAL_TO_WORD(CronEd.PR_TT*10));INTERN ASSIGN CronEd.PR.Setpoint[46]:=(REAL_TO_WORD(CronEd.PR_TT*10));INTERN ASSIGN CronEd.PR.Setpoint[45]:=(REAL_TO_WORD(CronEd.PR_TT*10));INTERN ASSIGN CronEd.PR.Setpoint[44]:=(REAL_TO_WORD(CronEd.PR_TT*10))
rectangle at (420,177)-(451,198): text "h12"; runs INTERN ASSIGN CronEd.PR.Setpoint[51]:=(REAL_TO_WORD(CronEd.PR_TT*10));INTERN ASSIGN CronEd.PR.Setpoint[50]:=(REAL_TO_WORD(CronEd.PR_TT*10));INTERN ASSIGN CronEd.PR.Setpoint[49]:=(REAL_TO_WORD(CronEd.PR_TT*10));INTERN ASSIGN CronEd.PR.Setpoint[48]:=(REAL_TO_WORD(CronEd.PR_TT*10))
rectangle at (450,177)-(481,198): text "h13"; runs INTERN ASSIGN CronEd.PR.Setpoint[55]:=(REAL_TO_WORD(CronEd.PR_TT*10));INTERN ASSIGN CronEd.PR.Setpoint[54]:=(REAL_TO_WORD(CronEd.PR_TT*10));INTERN ASSIGN CronEd.PR.Setpoint[53]:=(REAL_TO_WORD(CronEd.PR_TT*10));INTERN ASSIGN CronEd.PR.Setpoint[52]:=(REAL_TO_WORD(CronEd.PR_TT*10))
rectangle at (480,177)-(511,198): text "h14"; runs INTERN ASSIGN CronEd.PR.Setpoint[59]:=(REAL_TO_WORD(CronEd.PR_TT*10));INTERN ASSIGN CronEd.PR.Setpoint[58]:=(REAL_TO_WORD(CronEd.PR_TT*10));INTERN ASSIGN CronEd.PR.Setpoint[57]:=(REAL_TO_WORD(CronEd.PR_TT*10));INTERN ASSIGN CronEd.PR.Setpoint[56]:=(REAL_TO_WORD(CronEd.PR_TT*10))
rectangle at (510,177)-(541,198): text "h15"; runs INTERN ASSIGN CronEd.PR.Setpoint[63]:=(REAL_TO_WORD(CronEd.PR_TT*10));INTERN ASSIGN CronEd.PR.Setpoint[62]:=(REAL_TO_WORD(CronEd.PR_TT*10));INTERN ASSIGN CronEd.PR.Setpoint[61]:=(REAL_TO_WORD(CronEd.PR_TT*10));INTERN ASSIGN CronEd.PR.Setpoint[60]:=(REAL_TO_WORD(CronEd.PR_TT*10))
rectangle at (540,177)-(571,198): text "h16"; runs INTERN ASSIGN CronEd.PR.Setpoint[67]:=(REAL_TO_WORD(CronEd.PR_TT*10));INTERN ASSIGN CronEd.PR.Setpoint[66]:=(REAL_TO_WORD(CronEd.PR_TT*10));INTERN ASSIGN CronEd.PR.Setpoint[65]:=(REAL_TO_WORD(CronEd.PR_TT*10));INTERN ASSIGN CronEd.PR.Setpoint[64]:=(REAL_TO_WORD(CronEd.PR_TT*10))
rectangle at (570,177)-(601,198): text "h17"; runs INTERN ASSIGN CronEd.PR.Setpoint[71]:=(REAL_TO_WORD(CronEd.PR_TT*10));INTERN ASSIGN CronEd.PR.Setpoint[70]:=(REAL_TO_WORD(CronEd.PR_TT*10));INTERN ASSIGN CronEd.PR.Setpoint[69]:=(REAL_TO_WORD(CronEd.PR_TT*10));INTERN ASSIGN CronEd.PR.Setpoint[68]:=(REAL_TO_WORD(CronEd.PR_TT*10))
rectangle at (600,177)-(631,198): text "h18"; runs INTERN ASSIGN CronEd.PR.Setpoint[75]:=(REAL_TO_WORD(CronEd.PR_TT*10));INTERN ASSIGN CronEd.PR.Setpoint[74]:=(REAL_TO_WORD(CronEd.PR_TT*10));INTERN ASSIGN CronEd.PR.Setpoint[73]:=(REAL_TO_WORD(CronEd.PR_TT*10));INTERN ASSIGN CronEd.PR.Setpoint[72]:=(REAL_TO_WORD(CronEd.PR_TT*10))
rectangle at (630,177)-(661,198): text "h19"; runs INTERN ASSIGN CronEd.PR.Setpoint[79]:=(REAL_TO_WORD(CronEd.PR_TT*10));INTERN ASSIGN CronEd.PR.Setpoint[78]:=(REAL_TO_WORD(CronEd.PR_TT*10));INTERN ASSIGN CronEd.PR.Setpoint[77]:=(REAL_TO_WORD(CronEd.PR_TT*10));INTERN ASSIGN CronEd.PR.Setpoint[76]:=(REAL_TO_WORD(CronEd.PR_TT*10))
rectangle at (660,177)-(691,198): text "h20"; runs INTERN ASSIGN CronEd.PR.Setpoint[83]:=(REAL_TO_WORD(CronEd.PR_TT*10));INTERN ASSIGN CronEd.PR.Setpoint[82]:=(REAL_TO_WORD(CronEd.PR_TT*10));INTERN ASSIGN CronEd.PR.Setpoint[81]:=(REAL_TO_WORD(CronEd.PR_TT*10));INTERN ASSIGN CronEd.PR.Setpoint[80]:=(REAL_TO_WORD(CronEd.PR_TT*10))
rectangle at (690,177)-(721,198): text "h21"; runs INTERN ASSIGN CronEd.PR.Setpoint[87]:=(REAL_TO_WORD(CronEd.PR_TT*10));INTERN ASSIGN CronEd.PR.Setpoint[86]:=(REAL_TO_WORD(CronEd.PR_TT*10));INTERN ASSIGN CronEd.PR.Setpoint[85]:=(REAL_TO_WORD(CronEd.PR_TT*10));INTERN ASSIGN CronEd.PR.Setpoint[84]:=(REAL_TO_WORD(CronEd.PR_TT*10))
rectangle at (720,177)-(751,198): text "h22"; runs INTERN ASSIGN CronEd.PR.Setpoint[91]:=(REAL_TO_WORD(CronEd.PR_TT*10));INTERN ASSIGN CronEd.PR.Setpoint[90]:=(REAL_TO_WORD(CronEd.PR_TT*10));INTERN ASSIGN CronEd.PR.Setpoint[89]:=(REAL_TO_WORD(CronEd.PR_TT*10));INTERN ASSIGN CronEd.PR.Setpoint[88]:=(REAL_TO_WORD(CronEd.PR_TT*10))
rectangle at (750,177)-(781,198): text "h23"; runs INTERN ASSIGN CronEd.PR.Setpoint[95]:=(REAL_TO_WORD(CronEd.PR_TT*10));INTERN ASSIGN CronEd.PR.Setpoint[94]:=(REAL_TO_WORD(CronEd.PR_TT*10));INTERN ASSIGN CronEd.PR.Setpoint[93]:=(REAL_TO_WORD(CronEd.PR_TT*10));INTERN ASSIGN CronEd.PR.Setpoint[92]:=(REAL_TO_WORD(CronEd.PR_TT*10))
rectangle at (410,1152)-(491,1173): text "Month"
rectangle at (490,1152)-(531,1173): text "%d"; shows CronEd.CA_Sel; alarm colour if CronEd.CA_Sel<>CronEd.CA_Act; editable 1..12
rectangle at (410,1182)-(491,1203): text "Profile Nr."
rectangle at (490,1182)-(531,1203): text "%d"; shows CronEd.CA_TPR; editable 0..10
button at (540,1152)-(601,1173): text "Load"; toggles CronEd.CA_Load
button at (610,1152)-(671,1173): text "Save"; toggles CronEd.CA_Save
rounded rectangle at (160,1152)-(191,1173): text "%d"; shows CronEd.CA.Profile[0]; invisible if CronEd.CA_DayF>0; alarm colour if CronEd.CA.Profile[0]=0; runs INTERN ASSIGN CronEd.CA.Profile[0]:=(CronEd.CA_TPR)
rectangle at (120,1152)-(151,1173): text "1"
rounded rectangle at (190,1152)-(221,1173): text "%d"; shows CronEd.CA.Profile[1]; invisible if CronEd.CA_DayF>1; alarm colour if CronEd.CA.Profile[1]=0; runs INTERN ASSIGN CronEd.CA.Profile[1]:=(CronEd.CA_TPR)
rounded rectangle at (220,1152)-(251,1173): text "%d"; shows CronEd.CA.Profile[2]; invisible if CronEd.CA_DayF>2; alarm colour if CronEd.CA.Profile[2]=0; runs INTERN ASSIGN CronEd.CA.Profile[2]:=(CronEd.CA_TPR)
rounded rectangle at (250,1152)-(281,1173): text "%d"; shows CronEd.CA.Profile[3]; invisible if CronEd.CA_DayF>3; alarm colour if CronEd.CA.Profile[3]=0; runs INTERN ASSIGN CronEd.CA.Profile[3]:=(CronEd.CA_TPR)
rounded rectangle at (280,1152)-(311,1173): text "%d"; shows CronEd.CA.Profile[4]; invisible if CronEd.CA_DayF>4; alarm colour if CronEd.CA.Profile[4]=0; runs INTERN ASSIGN CronEd.CA.Profile[4]:=(CronEd.CA_TPR)
rounded rectangle at (310,1152)-(341,1173): text "%d"; shows CronEd.CA.Profile[5]; invisible if CronEd.CA_DayF>5; alarm colour if CronEd.CA.Profile[5]=0; runs INTERN ASSIGN CronEd.CA.Profile[5]:=(CronEd.CA_TPR)
rounded rectangle at (340,1152)-(371,1173): text "%d"; shows CronEd.CA.Profile[6]; alarm colour if CronEd.CA.Profile[6]=0; runs INTERN ASSIGN CronEd.CA.Profile[6]:=(CronEd.CA_TPR)
rounded rectangle at (160,1172)-(191,1193): text "%d"; shows CronEd.CA.Profile[7]; alarm colour if CronEd.CA.Profile[7]=0; runs INTERN ASSIGN CronEd.CA.Profile[7]:=(CronEd.CA_TPR)
rectangle at (120,1172)-(151,1193): text "8"
rounded rectangle at (190,1172)-(221,1193): text "%d"; shows CronEd.CA.Profile[8]; alarm colour if CronEd.CA.Profile[8]=0; runs INTERN ASSIGN CronEd.CA.Profile[8]:=(CronEd.CA_TPR)
rounded rectangle at (220,1172)-(251,1193): text "%d"; shows CronEd.CA.Profile[9]; alarm colour if CronEd.CA.Profile[9]=0; runs INTERN ASSIGN CronEd.CA.Profile[9]:=(CronEd.CA_TPR)
rounded rectangle at (250,1172)-(281,1193): text "%d"; shows CronEd.CA.Profile[10]; alarm colour if CronEd.CA.Profile[10]=0; runs INTERN ASSIGN CronEd.CA.Profile[10]:=(CronEd.CA_TPR)
rounded rectangle at (280,1172)-(311,1193): text "%d"; shows CronEd.CA.Profile[11]; alarm colour if CronEd.CA.Profile[11]=0; runs INTERN ASSIGN CronEd.CA.Profile[11]:=(CronEd.CA_TPR)
rounded rectangle at (310,1172)-(341,1193): text "%d"; shows CronEd.CA.Profile[12]; alarm colour if CronEd.CA.Profile[12]=0; runs INTERN ASSIGN CronEd.CA.Profile[12]:=(CronEd.CA_TPR)
rounded rectangle at (340,1172)-(371,1193): text "%d"; shows CronEd.CA.Profile[13]; alarm colour if CronEd.CA.Profile[13]=0; runs INTERN ASSIGN CronEd.CA.Profile[13]:=(CronEd.CA_TPR)
rounded rectangle at (160,1192)-(191,1213): text "%d"; shows CronEd.CA.Profile[14]; alarm colour if CronEd.CA.Profile[14]=0; runs INTERN ASSIGN CronEd.CA.Profile[14]:=(CronEd.CA_TPR)
rectangle at (120,1192)-(151,1213): text "15"
rounded rectangle at (190,1192)-(221,1213): text "%d"; shows CronEd.CA.Profile[15]; alarm colour if CronEd.CA.Profile[15]=0; runs INTERN ASSIGN CronEd.CA.Profile[15]:=(CronEd.CA_TPR)
rounded rectangle at (220,1192)-(251,1213): text "%d"; shows CronEd.CA.Profile[16]; alarm colour if CronEd.CA.Profile[16]=0; runs INTERN ASSIGN CronEd.CA.Profile[16]:=(CronEd.CA_TPR)
rounded rectangle at (250,1192)-(281,1213): text "%d"; shows CronEd.CA.Profile[17]; alarm colour if CronEd.CA.Profile[17]=0; runs INTERN ASSIGN CronEd.CA.Profile[17]:=(CronEd.CA_TPR)
rounded rectangle at (280,1192)-(311,1213): text "%d"; shows CronEd.CA.Profile[18]; alarm colour if CronEd.CA.Profile[18]=0; runs INTERN ASSIGN CronEd.CA.Profile[18]:=(CronEd.CA_TPR)
rounded rectangle at (310,1192)-(341,1213): text "%d"; shows CronEd.CA.Profile[19]; alarm colour if CronEd.CA.Profile[19]=0; runs INTERN ASSIGN CronEd.CA.Profile[19]:=(CronEd.CA_TPR)
rounded rectangle at (340,1192)-(371,1213): text "%d"; shows CronEd.CA.Profile[20]; alarm colour if CronEd.CA.Profile[20]=0; runs INTERN ASSIGN CronEd.CA.Profile[20]:=(CronEd.CA_TPR)
rounded rectangle at (160,1212)-(191,1233): text "%d"; shows CronEd.CA.Profile[21]; alarm colour if CronEd.CA.Profile[21]=0; runs INTERN ASSIGN CronEd.CA.Profile[21]:=(CronEd.CA_TPR)
rectangle at (120,1212)-(151,1233): text "22"
rounded rectangle at (190,1212)-(221,1233): text "%d"; shows CronEd.CA.Profile[22]; alarm colour if CronEd.CA.Profile[22]=0; runs INTERN ASSIGN CronEd.CA.Profile[22]:=(CronEd.CA_TPR)
rounded rectangle at (220,1212)-(251,1233): text "%d"; shows CronEd.CA.Profile[23]; alarm colour if CronEd.CA.Profile[23]=0; runs INTERN ASSIGN CronEd.CA.Profile[23]:=(CronEd.CA_TPR)
rounded rectangle at (250,1212)-(281,1233): text "%d"; shows CronEd.CA.Profile[24]; alarm colour if CronEd.CA.Profile[24]=0; runs INTERN ASSIGN CronEd.CA.Profile[24]:=(CronEd.CA_TPR)
rounded rectangle at (280,1212)-(311,1233): text "%d"; shows CronEd.CA.Profile[25]; alarm colour if CronEd.CA.Profile[25]=0; runs INTERN ASSIGN CronEd.CA.Profile[25]:=(CronEd.CA_TPR)
rounded rectangle at (310,1212)-(341,1233): text "%d"; shows CronEd.CA.Profile[26]; alarm colour if CronEd.CA.Profile[26]=0; runs INTERN ASSIGN CronEd.CA.Profile[26]:=(CronEd.CA_TPR)
rounded rectangle at (340,1212)-(371,1233): text "%d"; shows CronEd.CA.Profile[27]; alarm colour if CronEd.CA.Profile[27]=0; runs INTERN ASSIGN CronEd.CA.Profile[27]:=(CronEd.CA_TPR)
rounded rectangle at (160,1232)-(191,1253): text "%d"; shows CronEd.CA.Profile[28]; alarm colour if CronEd.CA.Profile[28]=0; runs INTERN ASSIGN CronEd.CA.Profile[28]:=(CronEd.CA_TPR)
rectangle at (120,1232)-(151,1253): text "29"
rounded rectangle at (190,1232)-(221,1253): text "%d"; shows CronEd.CA.Profile[29]; alarm colour if CronEd.CA.Profile[29]=0; runs INTERN ASSIGN CronEd.CA.Profile[29]:=(CronEd.CA_TPR)
rounded rectangle at (220,1232)-(251,1253): text "%d"; shows CronEd.CA.Profile[30]; alarm colour if CronEd.CA.Profile[30]=0; runs INTERN ASSIGN CronEd.CA.Profile[30]:=(CronEd.CA_TPR)
rounded rectangle at (250,1232)-(281,1253): text "%d"; shows CronEd.CA.Profile[31]; alarm colour if CronEd.CA.Profile[31]=0; runs INTERN ASSIGN CronEd.CA.Profile[31]:=(CronEd.CA_TPR)
rounded rectangle at (280,1232)-(311,1253): text "%d"; shows CronEd.CA.Profile[32]; invisible if CronEd.CA_DayL<32; alarm colour if CronEd.CA.Profile[32]=0; runs INTERN ASSIGN CronEd.CA.Profile[32]:=(CronEd.CA_TPR)
rounded rectangle at (310,1232)-(341,1253): text "%d"; shows CronEd.CA.Profile[33]; invisible if CronEd.CA_DayL<33; alarm colour if CronEd.CA.Profile[33]=0; runs INTERN ASSIGN CronEd.CA.Profile[33]:=(CronEd.CA_TPR)
rounded rectangle at (340,1232)-(371,1253): text "%d"; shows CronEd.CA.Profile[34]; invisible if CronEd.CA_DayL<34; alarm colour if CronEd.CA.Profile[34]=0; runs INTERN ASSIGN CronEd.CA.Profile[34]:=(CronEd.CA_TPR)
rounded rectangle at (160,1252)-(191,1273): text "%d"; shows CronEd.CA.Profile[35]; invisible if CronEd.CA_DayL<35; alarm colour if CronEd.CA.Profile[35]=0; runs INTERN ASSIGN CronEd.CA.Profile[35]:=(CronEd.CA_TPR)
rectangle at (120,1252)-(151,1273): text "36"; invisible if CronEd.CA_DayL<35
rounded rectangle at (190,1252)-(221,1273): text "%d"; shows CronEd.CA.Profile[36]; invisible if CronEd.CA_DayL<36; alarm colour if CronEd.CA.Profile[36]=0; runs INTERN ASSIGN CronEd.CA.Profile[36]:=(CronEd.CA_TPR)
rounded rectangle at (220,1252)-(251,1273): text "%d"; shows CronEd.CA.Profile[37]; invisible if CronEd.CA_DayL<37; alarm colour if CronEd.CA.Profile[37]=0; runs INTERN ASSIGN CronEd.CA.Profile[37]:=(CronEd.CA_TPR)
rounded rectangle at (250,1252)-(281,1273): text "%d"; shows CronEd.CA.Profile[38]; invisible if CronEd.CA_DayL<38; alarm colour if CronEd.CA.Profile[38]=0; runs INTERN ASSIGN CronEd.CA.Profile[38]:=(CronEd.CA_TPR)
rounded rectangle at (280,1252)-(311,1273): text "%d"; shows CronEd.CA.Profile[39]; invisible if CronEd.CA_DayL<39; alarm colour if CronEd.CA.Profile[39]=0; runs INTERN ASSIGN CronEd.CA.Profile[39]:=(CronEd.CA_TPR)
rounded rectangle at (310,1252)-(341,1273): text "%d"; shows CronEd.CA.Profile[40]; invisible if CronEd.CA_DayL<40; alarm colour if CronEd.CA.Profile[40]=0; runs INTERN ASSIGN CronEd.CA.Profile[40]:=(CronEd.CA_TPR)
rounded rectangle at (340,1252)-(371,1273): text "%d"; shows CronEd.CA.Profile[41]; invisible if CronEd.CA_DayL<41; alarm colour if CronEd.CA.Profile[41]=0; runs INTERN ASSIGN CronEd.CA.Profile[41]:=(CronEd.CA_TPR)
rectangle at (310,60)-(371,81): text "Year"
rectangle at (370,60)-(411,81): text "%d"; shows CronEd.CN_YSel; alarm colour if CronEd.CN_YSel<>CronEd.CN_YAct; editable 2000..2100
rectangle at (480,60)-(761,81): text "%s"; shows CronEd.Message
button at (10,50)-(71,81): text "REINIT"; runs INTERN ASSIGN CRON03.InitOK:=(FALSE);INTERN ASSIGN CRON04.InitOK:=(FALSE);INTERN ASSIGN CRON05.InitOK:=(FALSE);INTERN ASSIGN CRON06.InitOK:=(FALSE);INTERN ASSIGN CRON01.InitOK:=(FALSE)
rounded rectangle at (60,262)-(91,278): text "%.1f"; shows WORD_TO_REAL(CronEd.PR.Setpoint[4])/10; runs INTERN ASSIGN CronEd.PR.Setpoint[4]:=(REAL_TO_WORD(CronEd.PR_TT*10))
rounded rectangle at (60,277)-(91,293): text "%.1f"; shows WORD_TO_REAL(CronEd.PR.Setpoint[5])/10; runs INTERN ASSIGN CronEd.PR.Setpoint[5]:=(REAL_TO_WORD(CronEd.PR_TT*10))
rounded rectangle at (60,292)-(91,308): text "%.1f"; shows WORD_TO_REAL(CronEd.PR.Setpoint[6])/10; runs INTERN ASSIGN CronEd.PR.Setpoint[6]:=(REAL_TO_WORD(CronEd.PR_TT*10))
rounded rectangle at (60,307)-(91,323): text "%.1f"; shows WORD_TO_REAL(CronEd.PR.Setpoint[7])/10; runs INTERN ASSIGN CronEd.PR.Setpoint[7]:=(REAL_TO_WORD(CronEd.PR_TT*10))
rounded rectangle at (60,321)-(91,337): text "%.1f"; shows WORD_TO_REAL(CronEd.PR.Setpoint[8])/10; runs INTERN ASSIGN CronEd.PR.Setpoint[8]:=(REAL_TO_WORD(CronEd.PR_TT*10))
rounded rectangle at (60,336)-(91,352): text "%.1f"; shows WORD_TO_REAL(CronEd.PR.Setpoint[9])/10; runs INTERN ASSIGN CronEd.PR.Setpoint[9]:=(REAL_TO_WORD(CronEd.PR_TT*10))
rounded rectangle at (60,351)-(91,367): text "%.1f"; shows WORD_TO_REAL(CronEd.PR.Setpoint[10])/10; runs INTERN ASSIGN CronEd.PR.Setpoint[10]:=(REAL_TO_WORD(CronEd.PR_TT*10))
rounded rectangle at (60,366)-(91,382): text "%.1f"; shows WORD_TO_REAL(CronEd.PR.Setpoint[11])/10; runs INTERN ASSIGN CronEd.PR.Setpoint[11]:=(REAL_TO_WORD(CronEd.PR_TT*10))
rounded rectangle at (60,381)-(91,397): text "%.1f"; shows WORD_TO_REAL(CronEd.PR.Setpoint[12])/10; runs INTERN ASSIGN CronEd.PR.Setpoint[12]:=(REAL_TO_WORD(CronEd.PR_TT*10))
rounded rectangle at (60,396)-(91,412): text "%.1f"; shows WORD_TO_REAL(CronEd.PR.Setpoint[13])/10; runs INTERN ASSIGN CronEd.PR.Setpoint[13]:=(REAL_TO_WORD(CronEd.PR_TT*10))
rounded rectangle at (60,411)-(91,427): text "%.1f"; shows WORD_TO_REAL(CronEd.PR.Setpoint[14])/10; runs INTERN ASSIGN CronEd.PR.Setpoint[14]:=(REAL_TO_WORD(CronEd.PR_TT*10))
rounded rectangle at (60,426)-(91,442): text "%.1f"; shows WORD_TO_REAL(CronEd.PR.Setpoint[15])/10; runs INTERN ASSIGN CronEd.PR.Setpoint[15]:=(REAL_TO_WORD(CronEd.PR_TT*10))
rounded rectangle at (60,441)-(91,457): text "%.1f"; shows WORD_TO_REAL(CronEd.PR.Setpoint[16])/10; runs INTERN ASSIGN CronEd.PR.Setpoint[16]:=(REAL_TO_WORD(CronEd.PR_TT*10))
rounded rectangle at (60,456)-(91,472): text "%.1f"; shows WORD_TO_REAL(CronEd.PR.Setpoint[17])/10; runs INTERN ASSIGN CronEd.PR.Setpoint[17]:=(REAL_TO_WORD(CronEd.PR_TT*10))
rounded rectangle at (60,471)-(91,487): text "%.1f"; shows WORD_TO_REAL(CronEd.PR.Setpoint[18])/10; runs INTERN ASSIGN CronEd.PR.Setpoint[18]:=(REAL_TO_WORD(CronEd.PR_TT*10))
rounded rectangle at (60,486)-(91,502): text "%.1f"; shows WORD_TO_REAL(CronEd.PR.Setpoint[19])/10; runs INTERN ASSIGN CronEd.PR.Setpoint[19]:=(REAL_TO_WORD(CronEd.PR_TT*10))
rectangle at (20,262)-(51,278): text "m04"
rectangle at (20,277)-(51,293): text "m05"
rectangle at (20,292)-(51,308): text "m06"
rectangle at (20,307)-(51,323): text "m07"
rectangle at (20,321)-(51,337): text "m08"
rectangle at (20,336)-(51,352): text "m09"
rectangle at (20,351)-(51,367): text "m10"
rectangle at (20,366)-(51,382): text "m11"
rectangle at (20,380)-(51,396): text "m12"
rectangle at (20,395)-(51,411): text "m13"
rectangle at (20,410)-(51,426): text "m14"
rectangle at (20,425)-(51,441): text "m15"
rectangle at (20,439)-(51,455): text "m16"
rectangle at (20,454)-(51,470): text "m17"
rectangle at (20,469)-(51,485): text "m18"
rectangle at (20,484)-(51,500): text "m19"
rectangle at (20,498)-(51,514): text "m20"
rectangle at (20,513)-(51,529): text "m21"
rectangle at (20,528)-(51,544): text "m22"
rectangle at (20,543)-(51,559): text "m23"
rectangle at (20,557)-(51,573): text "m24"
rectangle at (20,572)-(51,588): text "m25"
rectangle at (20,587)-(51,603): text "m26"
rectangle at (20,602)-(51,618): text "m27"
rectangle at (21,616)-(52,632): text "m28"
rectangle at (21,631)-(52,647): text "m29"
rectangle at (21,646)-(52,662): text "m30"
rectangle at (21,661)-(52,677): text "m31"
rectangle at (21,675)-(52,691): text "m32"
rectangle at (21,690)-(52,706): text "m33"
rectangle at (21,705)-(52,721): text "m34"
rectangle at (21,720)-(52,736): text "m35"
rounded rectangle at (60,500)-(91,516): text "%.1f"; shows WORD_TO_REAL(CronEd.PR.Setpoint[20])/10; runs INTERN ASSIGN CronEd.PR.Setpoint[20]:=(REAL_TO_WORD(CronEd.PR_TT*10))
rounded rectangle at (60,515)-(91,531): text "%.1f"; shows WORD_TO_REAL(CronEd.PR.Setpoint[21])/10; runs INTERN ASSIGN CronEd.PR.Setpoint[21]:=(REAL_TO_WORD(CronEd.PR_TT*10))
rounded rectangle at (60,530)-(91,546): text "%.1f"; shows WORD_TO_REAL(CronEd.PR.Setpoint[22])/10; runs INTERN ASSIGN CronEd.PR.Setpoint[22]:=(REAL_TO_WORD(CronEd.PR_TT*10))
rounded rectangle at (60,545)-(91,561): text "%.1f"; shows WORD_TO_REAL(CronEd.PR.Setpoint[23])/10; runs INTERN ASSIGN CronEd.PR.Setpoint[23]:=(REAL_TO_WORD(CronEd.PR_TT*10))
rounded rectangle at (60,559)-(91,575): text "%.1f"; shows WORD_TO_REAL(CronEd.PR.Setpoint[24])/10; runs INTERN ASSIGN CronEd.PR.Setpoint[24]:=(REAL_TO_WORD(CronEd.PR_TT*10))
rounded rectangle at (60,574)-(91,590): text "%.1f"; shows WORD_TO_REAL(CronEd.PR.Setpoint[25])/10; runs INTERN ASSIGN CronEd.PR.Setpoint[25]:=(REAL_TO_WORD(CronEd.PR_TT*10))
rounded rectangle at (60,589)-(91,605): text "%.1f"; shows WORD_TO_REAL(CronEd.PR.Setpoint[26])/10; runs INTERN ASSIGN CronEd.PR.Setpoint[26]:=(REAL_TO_WORD(CronEd.PR_TT*10))
rounded rectangle at (60,604)-(91,620): text "%.1f"; shows WORD_TO_REAL(CronEd.PR.Setpoint[27])/10; runs INTERN ASSIGN CronEd.PR.Setpoint[27]:=(REAL_TO_WORD(CronEd.PR_TT*10))
rounded rectangle at (60,618)-(91,634): text "%.1f"; shows WORD_TO_REAL(CronEd.PR.Setpoint[28])/10; runs INTERN ASSIGN CronEd.PR.Setpoint[28]:=(REAL_TO_WORD(CronEd.PR_TT*10))
rounded rectangle at (60,633)-(91,649): text "%.1f"; shows WORD_TO_REAL(CronEd.PR.Setpoint[29])/10; runs INTERN ASSIGN CronEd.PR.Setpoint[29]:=(REAL_TO_WORD(CronEd.PR_TT*10))
rounded rectangle at (60,648)-(91,664): text "%.1f"; shows WORD_TO_REAL(CronEd.PR.Setpoint[30])/10; runs INTERN ASSIGN CronEd.PR.Setpoint[30]:=(REAL_TO_WORD(CronEd.PR_TT*10))
rounded rectangle at (60,663)-(91,679): text "%.1f"; shows WORD_TO_REAL(CronEd.PR.Setpoint[31])/10; runs INTERN ASSIGN CronEd.PR.Setpoint[31]:=(REAL_TO_WORD(CronEd.PR_TT*10))
rectangle at (21,735)-(52,751): text "m36"
rectangle at (21,750)-(52,766): text "m37"
rectangle at (21,764)-(52,780): text "m38"
rectangle at (21,779)-(52,795): text "m39"
rectangle at (21,794)-(52,810): text "m40"
rectangle at (21,809)-(52,825): text "m41"
rectangle at (21,824)-(52,840): text "m42"
rectangle at (21,839)-(52,855): text "m43"
rectangle at (21,854)-(52,870): text "m44"
rectangle at (21,869)-(52,885): text "m45"
rectangle at (21,884)-(52,900): text "m46"
rectangle at (21,899)-(52,915): text "m47"
rectangle at (21,915)-(52,931): text "m48"
rectangle at (21,930)-(52,946): text "m49"
rectangle at (21,945)-(52,961): text "m50"
rectangle at (21,960)-(52,976): text "m51"
rectangle at (21,975)-(52,991): text "m52"
rectangle at (21,990)-(52,1006): text "m53"
rectangle at (21,1005)-(52,1021): text "m54"
rectangle at (21,1020)-(52,1036): text "m55"
rectangle at (21,1035)-(52,1051): text "m56"
rectangle at (21,1050)-(52,1066): text "m57"
rectangle at (21,1066)-(52,1082): text "m58"
rectangle at (21,1081)-(52,1097): text "m59"
rounded rectangle at (60,677)-(91,693): text "%.1f"; shows WORD_TO_REAL(CronEd.PR.Setpoint[32])/10; runs INTERN ASSIGN CronEd.PR.Setpoint[32]:=(REAL_TO_WORD(CronEd.PR_TT*10))
rounded rectangle at (60,692)-(91,708): text "%.1f"; shows WORD_TO_REAL(CronEd.PR.Setpoint[33])/10; runs INTERN ASSIGN CronEd.PR.Setpoint[33]:=(REAL_TO_WORD(CronEd.PR_TT*10))
rounded rectangle at (60,707)-(91,723): text "%.1f"; shows WORD_TO_REAL(CronEd.PR.Setpoint[34])/10; runs INTERN ASSIGN CronEd.PR.Setpoint[34]:=(REAL_TO_WORD(CronEd.PR_TT*10))
rounded rectangle at (60,722)-(91,738): text "%.1f"; shows WORD_TO_REAL(CronEd.PR.Setpoint[35])/10; runs INTERN ASSIGN CronEd.PR.Setpoint[35]:=(REAL_TO_WORD(CronEd.PR_TT*10))
rounded rectangle at (60,737)-(91,753): text "%.1f"; shows WORD_TO_REAL(CronEd.PR.Setpoint[36])/10; runs INTERN ASSIGN CronEd.PR.Setpoint[36]:=(REAL_TO_WORD(CronEd.PR_TT*10))
rounded rectangle at (60,752)-(91,768): text "%.1f"; shows WORD_TO_REAL(CronEd.PR.Setpoint[37])/10; runs INTERN ASSIGN CronEd.PR.Setpoint[37]:=(REAL_TO_WORD(CronEd.PR_TT*10))
rounded rectangle at (60,767)-(91,783): text "%.1f"; shows WORD_TO_REAL(CronEd.PR.Setpoint[38])/10; runs INTERN ASSIGN CronEd.PR.Setpoint[38]:=(REAL_TO_WORD(CronEd.PR_TT*10))
rounded rectangle at (60,782)-(91,798): text "%.1f"; shows WORD_TO_REAL(CronEd.PR.Setpoint[39])/10; runs INTERN ASSIGN CronEd.PR.Setpoint[39]:=(REAL_TO_WORD(CronEd.PR_TT*10))
rounded rectangle at (60,796)-(91,812): text "%.1f"; shows WORD_TO_REAL(CronEd.PR.Setpoint[40])/10; runs INTERN ASSIGN CronEd.PR.Setpoint[40]:=(REAL_TO_WORD(CronEd.PR_TT*10))
rounded rectangle at (60,811)-(91,827): text "%.1f"; shows WORD_TO_REAL(CronEd.PR.Setpoint[41])/10; runs INTERN ASSIGN CronEd.PR.Setpoint[41]:=(REAL_TO_WORD(CronEd.PR_TT*10))
rounded rectangle at (60,826)-(91,842): text "%.1f"; shows WORD_TO_REAL(CronEd.PR.Setpoint[42])/10; runs INTERN ASSIGN CronEd.PR.Setpoint[42]:=(REAL_TO_WORD(CronEd.PR_TT*10))
rounded rectangle at (60,841)-(91,857): text "%.1f"; shows WORD_TO_REAL(CronEd.PR.Setpoint[43])/10; runs INTERN ASSIGN CronEd.PR.Setpoint[43]:=(REAL_TO_WORD(CronEd.PR_TT*10))
rounded rectangle at (60,855)-(91,871): text "%.1f"; shows WORD_TO_REAL(CronEd.PR.Setpoint[44])/10; runs INTERN ASSIGN CronEd.PR.Setpoint[44]:=(REAL_TO_WORD(CronEd.PR_TT*10))
rounded rectangle at (60,870)-(91,886): text "%.1f"; shows WORD_TO_REAL(CronEd.PR.Setpoint[45])/10; runs INTERN ASSIGN CronEd.PR.Setpoint[45]:=(REAL_TO_WORD(CronEd.PR_TT*10))
rounded rectangle at (60,885)-(91,901): text "%.1f"; shows WORD_TO_REAL(CronEd.PR.Setpoint[46])/10; runs INTERN ASSIGN CronEd.PR.Setpoint[46]:=(REAL_TO_WORD(CronEd.PR_TT*10))
rounded rectangle at (60,900)-(91,916): text "%.1f"; shows WORD_TO_REAL(CronEd.PR.Setpoint[47])/10; runs INTERN ASSIGN CronEd.PR.Setpoint[47]:=(REAL_TO_WORD(CronEd.PR_TT*10))
rounded rectangle at (59,914)-(90,930): text "%.1f"; shows WORD_TO_REAL(CronEd.PR.Setpoint[48])/10; runs INTERN ASSIGN CronEd.PR.Setpoint[48]:=(REAL_TO_WORD(CronEd.PR_TT*10))
rounded rectangle at (59,929)-(90,945): text "%.1f"; shows WORD_TO_REAL(CronEd.PR.Setpoint[49])/10; runs INTERN ASSIGN CronEd.PR.Setpoint[49]:=(REAL_TO_WORD(CronEd.PR_TT*10))
rounded rectangle at (59,944)-(90,960): text "%.1f"; shows WORD_TO_REAL(CronEd.PR.Setpoint[50])/10; runs INTERN ASSIGN CronEd.PR.Setpoint[50]:=(REAL_TO_WORD(CronEd.PR_TT*10))
rounded rectangle at (59,959)-(90,975): text "%.1f"; shows WORD_TO_REAL(CronEd.PR.Setpoint[51])/10; runs INTERN ASSIGN CronEd.PR.Setpoint[51]:=(REAL_TO_WORD(CronEd.PR_TT*10))
rounded rectangle at (58,973)-(89,989): text "%.1f"; shows WORD_TO_REAL(CronEd.PR.Setpoint[52])/10; runs INTERN ASSIGN CronEd.PR.Setpoint[52]:=(REAL_TO_WORD(CronEd.PR_TT*10))
rounded rectangle at (58,988)-(89,1004): text "%.1f"; shows WORD_TO_REAL(CronEd.PR.Setpoint[53])/10; runs INTERN ASSIGN CronEd.PR.Setpoint[53]:=(REAL_TO_WORD(CronEd.PR_TT*10))
rounded rectangle at (58,1003)-(89,1019): text "%.1f"; shows WORD_TO_REAL(CronEd.PR.Setpoint[54])/10; runs INTERN ASSIGN CronEd.PR.Setpoint[54]:=(REAL_TO_WORD(CronEd.PR_TT*10))
rounded rectangle at (58,1018)-(89,1034): text "%.1f"; shows WORD_TO_REAL(CronEd.PR.Setpoint[55])/10; runs INTERN ASSIGN CronEd.PR.Setpoint[55]:=(REAL_TO_WORD(CronEd.PR_TT*10))
rounded rectangle at (57,1033)-(88,1049): text "%.1f"; shows WORD_TO_REAL(CronEd.PR.Setpoint[56])/10; runs INTERN ASSIGN CronEd.PR.Setpoint[56]:=(REAL_TO_WORD(CronEd.PR_TT*10))
rounded rectangle at (57,1048)-(88,1064): text "%.1f"; shows WORD_TO_REAL(CronEd.PR.Setpoint[57])/10; runs INTERN ASSIGN CronEd.PR.Setpoint[57]:=(REAL_TO_WORD(CronEd.PR_TT*10))
rounded rectangle at (57,1063)-(88,1079): text "%.1f"; shows WORD_TO_REAL(CronEd.PR.Setpoint[58])/10; runs INTERN ASSIGN CronEd.PR.Setpoint[58]:=(REAL_TO_WORD(CronEd.PR_TT*10))
rounded rectangle at (57,1078)-(88,1094): text "%.1f"; shows WORD_TO_REAL(CronEd.PR.Setpoint[59])/10; runs INTERN ASSIGN CronEd.PR.Setpoint[59]:=(REAL_TO_WORD(CronEd.PR_TT*10))
rounded rectangle at (90,203)-(121,219): text "%.1f"; shows WORD_TO_REAL(CronEd.PR.Setpoint[60])/10; runs INTERN ASSIGN CronEd.PR.Setpoint[60]:=(REAL_TO_WORD(CronEd.PR_TT*10))
rounded rectangle at (90,218)-(121,234): text "%.1f"; shows WORD_TO_REAL(CronEd.PR.Setpoint[61])/10; runs INTERN ASSIGN CronEd.PR.Setpoint[61]:=(REAL_TO_WORD(CronEd.PR_TT*10))
rounded rectangle at (90,233)-(121,249): text "%.1f"; shows WORD_TO_REAL(CronEd.PR.Setpoint[62])/10; runs INTERN ASSIGN CronEd.PR.Setpoint[62]:=(REAL_TO_WORD(CronEd.PR_TT*10))
rounded rectangle at (90,248)-(121,264): text "%.1f"; shows WORD_TO_REAL(CronEd.PR.Setpoint[63])/10; runs INTERN ASSIGN CronEd.PR.Setpoint[63]:=(REAL_TO_WORD(CronEd.PR_TT*10))
rounded rectangle at (90,262)-(121,278): text "%.1f"; shows WORD_TO_REAL(CronEd.PR.Setpoint[64])/10; runs INTERN ASSIGN CronEd.PR.Setpoint[64]:=(REAL_TO_WORD(CronEd.PR_TT*10))
rounded rectangle at (90,277)-(121,293): text "%.1f"; shows WORD_TO_REAL(CronEd.PR.Setpoint[65])/10; runs INTERN ASSIGN CronEd.PR.Setpoint[65]:=(REAL_TO_WORD(CronEd.PR_TT*10))
rounded rectangle at (90,292)-(121,308): text "%.1f"; shows WORD_TO_REAL(CronEd.PR.Setpoint[66])/10; runs INTERN ASSIGN CronEd.PR.Setpoint[66]:=(REAL_TO_WORD(CronEd.PR_TT*10))
rounded rectangle at (90,307)-(121,323): text "%.1f"; shows WORD_TO_REAL(CronEd.PR.Setpoint[67])/10; runs INTERN ASSIGN CronEd.PR.Setpoint[67]:=(REAL_TO_WORD(CronEd.PR_TT*10))
rounded rectangle at (90,321)-(121,337): text "%.1f"; shows WORD_TO_REAL(CronEd.PR.Setpoint[68])/10; runs INTERN ASSIGN CronEd.PR.Setpoint[68]:=(REAL_TO_WORD(CronEd.PR_TT*10))
rounded rectangle at (90,336)-(121,352): text "%.1f"; shows WORD_TO_REAL(CronEd.PR.Setpoint[69])/10; runs INTERN ASSIGN CronEd.PR.Setpoint[69]:=(REAL_TO_WORD(CronEd.PR_TT*10))
rounded rectangle at (90,351)-(121,367): text "%.1f"; shows WORD_TO_REAL(CronEd.PR.Setpoint[70])/10; runs INTERN ASSIGN CronEd.PR.Setpoint[70]:=(REAL_TO_WORD(CronEd.PR_TT*10))
rounded rectangle at (90,366)-(121,382): text "%.1f"; shows WORD_TO_REAL(CronEd.PR.Setpoint[71])/10; runs INTERN ASSIGN CronEd.PR.Setpoint[71]:=(REAL_TO_WORD(CronEd.PR_TT*10))
rounded rectangle at (90,380)-(121,396): text "%.1f"; shows WORD_TO_REAL(CronEd.PR.Setpoint[72])/10; runs INTERN ASSIGN CronEd.PR.Setpoint[72]:=(REAL_TO_WORD(CronEd.PR_TT*10))
rounded rectangle at (90,395)-(121,411): text "%.1f"; shows WORD_TO_REAL(CronEd.PR.Setpoint[73])/10; runs INTERN ASSIGN CronEd.PR.Setpoint[73]:=(REAL_TO_WORD(CronEd.PR_TT*10))
rounded rectangle at (90,410)-(121,426): text "%.1f"; shows WORD_TO_REAL(CronEd.PR.Setpoint[74])/10; runs INTERN ASSIGN CronEd.PR.Setpoint[74]:=(REAL_TO_WORD(CronEd.PR_TT*10))
rounded rectangle at (90,425)-(121,441): text "%.1f"; shows WORD_TO_REAL(CronEd.PR.Setpoint[75])/10; runs INTERN ASSIGN CronEd.PR.Setpoint[75]:=(REAL_TO_WORD(CronEd.PR_TT*10))
rounded rectangle at (90,440)-(121,456): text "%.1f"; shows WORD_TO_REAL(CronEd.PR.Setpoint[76])/10; runs INTERN ASSIGN CronEd.PR.Setpoint[76]:=(REAL_TO_WORD(CronEd.PR_TT*10))
rounded rectangle at (90,455)-(121,471): text "%.1f"; shows WORD_TO_REAL(CronEd.PR.Setpoint[77])/10; runs INTERN ASSIGN CronEd.PR.Setpoint[77]:=(REAL_TO_WORD(CronEd.PR_TT*10))
rounded rectangle at (90,470)-(121,486): text "%.1f"; shows WORD_TO_REAL(CronEd.PR.Setpoint[78])/10; runs INTERN ASSIGN CronEd.PR.Setpoint[78]:=(REAL_TO_WORD(CronEd.PR_TT*10))
rounded rectangle at (90,485)-(121,501): text "%.1f"; shows WORD_TO_REAL(CronEd.PR.Setpoint[79])/10; runs INTERN ASSIGN CronEd.PR.Setpoint[79]:=(REAL_TO_WORD(CronEd.PR_TT*10))
rounded rectangle at (90,499)-(121,515): text "%.1f"; shows WORD_TO_REAL(CronEd.PR.Setpoint[80])/10; runs INTERN ASSIGN CronEd.PR.Setpoint[80]:=(REAL_TO_WORD(CronEd.PR_TT*10))
rounded rectangle at (90,514)-(121,530): text "%.1f"; shows WORD_TO_REAL(CronEd.PR.Setpoint[81])/10; runs INTERN ASSIGN CronEd.PR.Setpoint[81]:=(REAL_TO_WORD(CronEd.PR_TT*10))
rounded rectangle at (90,529)-(121,545): text "%.1f"; shows WORD_TO_REAL(CronEd.PR.Setpoint[82])/10; runs INTERN ASSIGN CronEd.PR.Setpoint[82]:=(REAL_TO_WORD(CronEd.PR_TT*10))
rounded rectangle at (90,544)-(121,560): text "%.1f"; shows WORD_TO_REAL(CronEd.PR.Setpoint[83])/10; runs INTERN ASSIGN CronEd.PR.Setpoint[83]:=(REAL_TO_WORD(CronEd.PR_TT*10))
rounded rectangle at (90,558)-(121,574): text "%.1f"; shows WORD_TO_REAL(CronEd.PR.Setpoint[84])/10; runs INTERN ASSIGN CronEd.PR.Setpoint[84]:=(REAL_TO_WORD(CronEd.PR_TT*10))
rounded rectangle at (90,573)-(121,589): text "%.1f"; shows WORD_TO_REAL(CronEd.PR.Setpoint[85])/10; runs INTERN ASSIGN CronEd.PR.Setpoint[85]:=(REAL_TO_WORD(CronEd.PR_TT*10))
rounded rectangle at (90,588)-(121,604): text "%.1f"; shows WORD_TO_REAL(CronEd.PR.Setpoint[86])/10; runs INTERN ASSIGN CronEd.PR.Setpoint[86]:=(REAL_TO_WORD(CronEd.PR_TT*10))
rounded rectangle at (90,603)-(121,619): text "%.1f"; shows WORD_TO_REAL(CronEd.PR.Setpoint[87])/10; runs INTERN ASSIGN CronEd.PR.Setpoint[87]:=(REAL_TO_WORD(CronEd.PR_TT*10))
rounded rectangle at (90,617)-(121,633): text "%.1f"; shows WORD_TO_REAL(CronEd.PR.Setpoint[88])/10; runs INTERN ASSIGN CronEd.PR.Setpoint[88]:=(REAL_TO_WORD(CronEd.PR_TT*10))
rounded rectangle at (90,632)-(121,648): text "%.1f"; shows WORD_TO_REAL(CronEd.PR.Setpoint[89])/10; runs INTERN ASSIGN CronEd.PR.Setpoint[89]:=(REAL_TO_WORD(CronEd.PR_TT*10))
rounded rectangle at (90,647)-(121,663): text "%.1f"; shows WORD_TO_REAL(CronEd.PR.Setpoint[90])/10; runs INTERN ASSIGN CronEd.PR.Setpoint[90]:=(REAL_TO_WORD(CronEd.PR_TT*10))
rounded rectangle at (90,662)-(121,678): text "%.1f"; shows WORD_TO_REAL(CronEd.PR.Setpoint[91])/10; runs INTERN ASSIGN CronEd.PR.Setpoint[91]:=(REAL_TO_WORD(CronEd.PR_TT*10))
rounded rectangle at (90,676)-(121,692): text "%.1f"; shows WORD_TO_REAL(CronEd.PR.Setpoint[92])/10; runs INTERN ASSIGN CronEd.PR.Setpoint[92]:=(REAL_TO_WORD(CronEd.PR_TT*10))
rounded rectangle at (90,691)-(121,707): text "%.1f"; shows WORD_TO_REAL(CronEd.PR.Setpoint[93])/10; runs INTERN ASSIGN CronEd.PR.Setpoint[93]:=(REAL_TO_WORD(CronEd.PR_TT*10))
rounded rectangle at (90,706)-(121,722): text "%.1f"; shows WORD_TO_REAL(CronEd.PR.Setpoint[94])/10; runs INTERN ASSIGN CronEd.PR.Setpoint[94]:=(REAL_TO_WORD(CronEd.PR_TT*10))
rounded rectangle at (90,721)-(121,737): text "%.1f"; shows WORD_TO_REAL(CronEd.PR.Setpoint[95])/10; runs INTERN ASSIGN CronEd.PR.Setpoint[95]:=(REAL_TO_WORD(CronEd.PR_TT*10))
rounded rectangle at (90,736)-(121,752): text "%.1f"; shows WORD_TO_REAL(CronEd.PR.Setpoint[96])/10; runs INTERN ASSIGN CronEd.PR.Setpoint[96]:=(REAL_TO_WORD(CronEd.PR_TT*10))
rounded rectangle at (90,751)-(121,767): text "%.1f"; shows WORD_TO_REAL(CronEd.PR.Setpoint[97])/10; runs INTERN ASSIGN CronEd.PR.Setpoint[97]:=(REAL_TO_WORD(CronEd.PR_TT*10))
rounded rectangle at (90,766)-(121,782): text "%.1f"; shows WORD_TO_REAL(CronEd.PR.Setpoint[98])/10; runs INTERN ASSIGN CronEd.PR.Setpoint[98]:=(REAL_TO_WORD(CronEd.PR_TT*10))
rounded rectangle at (90,781)-(121,797): text "%.1f"; shows WORD_TO_REAL(CronEd.PR.Setpoint[99])/10; runs INTERN ASSIGN CronEd.PR.Setpoint[99]:=(REAL_TO_WORD(CronEd.PR_TT*10))
rounded rectangle at (90,795)-(121,811): text "%.1f"; shows WORD_TO_REAL(CronEd.PR.Setpoint[100])/10; runs INTERN ASSIGN CronEd.PR.Setpoint[100]:=(REAL_TO_WORD(CronEd.PR_TT*10))
rounded rectangle at (90,810)-(121,826): text "%.1f"; shows WORD_TO_REAL(CronEd.PR.Setpoint[101])/10; runs INTERN ASSIGN CronEd.PR.Setpoint[101]:=(REAL_TO_WORD(CronEd.PR_TT*10))
rounded rectangle at (90,825)-(121,841): text "%.1f"; shows WORD_TO_REAL(CronEd.PR.Setpoint[102])/10; runs INTERN ASSIGN CronEd.PR.Setpoint[102]:=(REAL_TO_WORD(CronEd.PR_TT*10))
rounded rectangle at (90,840)-(121,856): text "%.1f"; shows WORD_TO_REAL(CronEd.PR.Setpoint[103])/10; runs INTERN ASSIGN CronEd.PR.Setpoint[103]:=(REAL_TO_WORD(CronEd.PR_TT*10))
rounded rectangle at (90,854)-(121,870): text "%.1f"; shows WORD_TO_REAL(CronEd.PR.Setpoint[104])/10; runs INTERN ASSIGN CronEd.PR.Setpoint[104]:=(REAL_TO_WORD(CronEd.PR_TT*10))
rounded rectangle at (90,869)-(121,885): text "%.1f"; shows WORD_TO_REAL(CronEd.PR.Setpoint[105])/10; runs INTERN ASSIGN CronEd.PR.Setpoint[105]:=(REAL_TO_WORD(CronEd.PR_TT*10))
rounded rectangle at (90,884)-(121,900): text "%.1f"; shows WORD_TO_REAL(CronEd.PR.Setpoint[106])/10; runs INTERN ASSIGN CronEd.PR.Setpoint[106]:=(REAL_TO_WORD(CronEd.PR_TT*10))
rounded rectangle at (90,899)-(121,915): text "%.1f"; shows WORD_TO_REAL(CronEd.PR.Setpoint[107])/10; runs INTERN ASSIGN CronEd.PR.Setpoint[107]:=(REAL_TO_WORD(CronEd.PR_TT*10))
rounded rectangle at (90,913)-(121,929): text "%.1f"; shows WORD_TO_REAL(CronEd.PR.Setpoint[108])/10; runs INTERN ASSIGN CronEd.PR.Setpoint[108]:=(REAL_TO_WORD(CronEd.PR_TT*10))
rounded rectangle at (90,928)-(121,944): text "%.1f"; shows WORD_TO_REAL(CronEd.PR.Setpoint[109])/10; runs INTERN ASSIGN CronEd.PR.Setpoint[109]:=(REAL_TO_WORD(CronEd.PR_TT*10))
rounded rectangle at (90,943)-(121,959): text "%.1f"; shows WORD_TO_REAL(CronEd.PR.Setpoint[110])/10; runs INTERN ASSIGN CronEd.PR.Setpoint[110]:=(REAL_TO_WORD(CronEd.PR_TT*10))
rounded rectangle at (90,958)-(121,974): text "%.1f"; shows WORD_TO_REAL(CronEd.PR.Setpoint[111])/10; runs INTERN ASSIGN CronEd.PR.Setpoint[111]:=(REAL_TO_WORD(CronEd.PR_TT*10))
rounded rectangle at (90,972)-(121,988): text "%.1f"; shows WORD_TO_REAL(CronEd.PR.Setpoint[112])/10; runs INTERN ASSIGN CronEd.PR.Setpoint[112]:=(REAL_TO_WORD(CronEd.PR_TT*10))
rounded rectangle at (90,987)-(121,1003): text "%.1f"; shows WORD_TO_REAL(CronEd.PR.Setpoint[113])/10; runs INTERN ASSIGN CronEd.PR.Setpoint[113]:=(REAL_TO_WORD(CronEd.PR_TT*10))
rounded rectangle at (90,1002)-(121,1018): text "%.1f"; shows WORD_TO_REAL(CronEd.PR.Setpoint[114])/10; runs INTERN ASSIGN CronEd.PR.Setpoint[114]:=(REAL_TO_WORD(CronEd.PR_TT*10))
rounded rectangle at (90,1017)-(121,1033): text "%.1f"; shows WORD_TO_REAL(CronEd.PR.Setpoint[115])/10; runs INTERN ASSIGN CronEd.PR.Setpoint[115]:=(REAL_TO_WORD(CronEd.PR_TT*10))
rounded rectangle at (90,1032)-(121,1048): text "%.1f"; shows WORD_TO_REAL(CronEd.PR.Setpoint[116])/10; runs INTERN ASSIGN CronEd.PR.Setpoint[116]:=(REAL_TO_WORD(CronEd.PR_TT*10))
rounded rectangle at (90,1047)-(121,1063): text "%.1f"; shows WORD_TO_REAL(CronEd.PR.Setpoint[117])/10; runs INTERN ASSIGN CronEd.PR.Setpoint[117]:=(REAL_TO_WORD(CronEd.PR_TT*10))
rounded rectangle at (90,1062)-(121,1078): text "%.1f"; shows WORD_TO_REAL(CronEd.PR.Setpoint[118])/10; runs INTERN ASSIGN CronEd.PR.Setpoint[118]:=(REAL_TO_WORD(CronEd.PR_TT*10))
rounded rectangle at (90,1077)-(121,1093): text "%.1f"; shows WORD_TO_REAL(CronEd.PR.Setpoint[119])/10; runs INTERN ASSIGN CronEd.PR.Setpoint[119]:=(REAL_TO_WORD(CronEd.PR_TT*10))
rounded rectangle at (120,203)-(151,219): text "%.1f"; shows WORD_TO_REAL(CronEd.PR.Setpoint[120])/10; runs INTERN ASSIGN CronEd.PR.Setpoint[120]:=(REAL_TO_WORD(CronEd.PR_TT*10))
rounded rectangle at (120,218)-(151,234): text "%.1f"; shows WORD_TO_REAL(CronEd.PR.Setpoint[121])/10; runs INTERN ASSIGN CronEd.PR.Setpoint[121]:=(REAL_TO_WORD(CronEd.PR_TT*10))
rounded rectangle at (120,233)-(151,249): text "%.1f"; shows WORD_TO_REAL(CronEd.PR.Setpoint[122])/10; runs INTERN ASSIGN CronEd.PR.Setpoint[122]:=(REAL_TO_WORD(CronEd.PR_TT*10))
rounded rectangle at (120,248)-(151,264): text "%.1f"; shows WORD_TO_REAL(CronEd.PR.Setpoint[123])/10; runs INTERN ASSIGN CronEd.PR.Setpoint[123]:=(REAL_TO_WORD(CronEd.PR_TT*10))
rounded rectangle at (120,262)-(151,278): text "%.1f"; shows WORD_TO_REAL(CronEd.PR.Setpoint[124])/10; runs INTERN ASSIGN CronEd.PR.Setpoint[124]:=(REAL_TO_WORD(CronEd.PR_TT*10))
rounded rectangle at (120,277)-(151,293): text "%.1f"; shows WORD_TO_REAL(CronEd.PR.Setpoint[125])/10; runs INTERN ASSIGN CronEd.PR.Setpoint[125]:=(REAL_TO_WORD(CronEd.PR_TT*10))
rounded rectangle at (120,292)-(151,308): text "%.1f"; shows WORD_TO_REAL(CronEd.PR.Setpoint[126])/10; runs INTERN ASSIGN CronEd.PR.Setpoint[126]:=(REAL_TO_WORD(CronEd.PR_TT*10))
rounded rectangle at (120,307)-(151,323): text "%.1f"; shows WORD_TO_REAL(CronEd.PR.Setpoint[127])/10; runs INTERN ASSIGN CronEd.PR.Setpoint[127]:=(REAL_TO_WORD(CronEd.PR_TT*10))
rounded rectangle at (120,321)-(151,337): text "%.1f"; shows WORD_TO_REAL(CronEd.PR.Setpoint[128])/10; runs INTERN ASSIGN CronEd.PR.Setpoint[128]:=(REAL_TO_WORD(CronEd.PR_TT*10))
rounded rectangle at (120,336)-(151,352): text "%.1f"; shows WORD_TO_REAL(CronEd.PR.Setpoint[129])/10; runs INTERN ASSIGN CronEd.PR.Setpoint[129]:=(REAL_TO_WORD(CronEd.PR_TT*10))
rounded rectangle at (120,351)-(151,367): text "%.1f"; shows WORD_TO_REAL(CronEd.PR.Setpoint[130])/10; runs INTERN ASSIGN CronEd.PR.Setpoint[130]:=(REAL_TO_WORD(CronEd.PR_TT*10))
rounded rectangle at (120,366)-(151,382): text "%.1f"; shows WORD_TO_REAL(CronEd.PR.Setpoint[131])/10; runs INTERN ASSIGN CronEd.PR.Setpoint[131]:=(REAL_TO_WORD(CronEd.PR_TT*10))
rounded rectangle at (120,380)-(151,396): text "%.1f"; shows WORD_TO_REAL(CronEd.PR.Setpoint[132])/10; runs INTERN ASSIGN CronEd.PR.Setpoint[132]:=(REAL_TO_WORD(CronEd.PR_TT*10))
rounded rectangle at (120,395)-(151,411): text "%.1f"; shows WORD_TO_REAL(CronEd.PR.Setpoint[133])/10; runs INTERN ASSIGN CronEd.PR.Setpoint[133]:=(REAL_TO_WORD(CronEd.PR_TT*10))
rounded rectangle at (120,410)-(151,426): text "%.1f"; shows WORD_TO_REAL(CronEd.PR.Setpoint[134])/10; runs INTERN ASSIGN CronEd.PR.Setpoint[134]:=(REAL_TO_WORD(CronEd.PR_TT*10))
rounded rectangle at (120,425)-(151,441): text "%.1f"; shows WORD_TO_REAL(CronEd.PR.Setpoint[135])/10; runs INTERN ASSIGN CronEd.PR.Setpoint[135]:=(REAL_TO_WORD(CronEd.PR_TT*10))
rounded rectangle at (120,440)-(151,456): text "%.1f"; shows WORD_TO_REAL(CronEd.PR.Setpoint[136])/10; runs INTERN ASSIGN CronEd.PR.Setpoint[136]:=(REAL_TO_WORD(CronEd.PR_TT*10))
rounded rectangle at (120,455)-(151,471): text "%.1f"; shows WORD_TO_REAL(CronEd.PR.Setpoint[137])/10; runs INTERN ASSIGN CronEd.PR.Setpoint[137]:=(REAL_TO_WORD(CronEd.PR_TT*10))
rounded rectangle at (120,470)-(151,486): text "%.1f"; shows WORD_TO_REAL(CronEd.PR.Setpoint[138])/10; runs INTERN ASSIGN CronEd.PR.Setpoint[138]:=(REAL_TO_WORD(CronEd.PR_TT*10))
rounded rectangle at (120,485)-(151,501): text "%.1f"; shows WORD_TO_REAL(CronEd.PR.Setpoint[139])/10; runs INTERN ASSIGN CronEd.PR.Setpoint[139]:=(REAL_TO_WORD(CronEd.PR_TT*10))
rounded rectangle at (120,499)-(151,515): text "%.1f"; shows WORD_TO_REAL(CronEd.PR.Setpoint[140])/10; runs INTERN ASSIGN CronEd.PR.Setpoint[140]:=(REAL_TO_WORD(CronEd.PR_TT*10))
rounded rectangle at (120,514)-(151,530): text "%.1f"; shows WORD_TO_REAL(CronEd.PR.Setpoint[141])/10; runs INTERN ASSIGN CronEd.PR.Setpoint[141]:=(REAL_TO_WORD(CronEd.PR_TT*10))
rounded rectangle at (120,529)-(151,545): text "%.1f"; shows WORD_TO_REAL(CronEd.PR.Setpoint[142])/10; runs INTERN ASSIGN CronEd.PR.Setpoint[142]:=(REAL_TO_WORD(CronEd.PR_TT*10))
rounded rectangle at (120,544)-(151,560): text "%.1f"; shows WORD_TO_REAL(CronEd.PR.Setpoint[143])/10; runs INTERN ASSIGN CronEd.PR.Setpoint[143]:=(REAL_TO_WORD(CronEd.PR_TT*10))
rounded rectangle at (120,558)-(151,574): text "%.1f"; shows WORD_TO_REAL(CronEd.PR.Setpoint[144])/10; runs INTERN ASSIGN CronEd.PR.Setpoint[144]:=(REAL_TO_WORD(CronEd.PR_TT*10))
rounded rectangle at (120,573)-(151,589): text "%.1f"; shows WORD_TO_REAL(CronEd.PR.Setpoint[145])/10; runs INTERN ASSIGN CronEd.PR.Setpoint[145]:=(REAL_TO_WORD(CronEd.PR_TT*10))
rounded rectangle at (120,588)-(151,604): text "%.1f"; shows WORD_TO_REAL(CronEd.PR.Setpoint[146])/10; runs INTERN ASSIGN CronEd.PR.Setpoint[146]:=(REAL_TO_WORD(CronEd.PR_TT*10))
rounded rectangle at (120,603)-(151,619): text "%.1f"; shows WORD_TO_REAL(CronEd.PR.Setpoint[147])/10; runs INTERN ASSIGN CronEd.PR.Setpoint[147]:=(REAL_TO_WORD(CronEd.PR_TT*10))
rounded rectangle at (120,617)-(151,633): text "%.1f"; shows WORD_TO_REAL(CronEd.PR.Setpoint[148])/10; runs INTERN ASSIGN CronEd.PR.Setpoint[148]:=(REAL_TO_WORD(CronEd.PR_TT*10))
rounded rectangle at (120,632)-(151,648): text "%.1f"; shows WORD_TO_REAL(CronEd.PR.Setpoint[149])/10; runs INTERN ASSIGN CronEd.PR.Setpoint[149]:=(REAL_TO_WORD(CronEd.PR_TT*10))
rounded rectangle at (120,647)-(151,663): text "%.1f"; shows WORD_TO_REAL(CronEd.PR.Setpoint[150])/10; runs INTERN ASSIGN CronEd.PR.Setpoint[150]:=(REAL_TO_WORD(CronEd.PR_TT*10))
rounded rectangle at (120,662)-(151,678): text "%.1f"; shows WORD_TO_REAL(CronEd.PR.Setpoint[151])/10; runs INTERN ASSIGN CronEd.PR.Setpoint[151]:=(REAL_TO_WORD(CronEd.PR_TT*10))
rounded rectangle at (570,677)-(601,693): text "%.1f"; shows WORD_TO_REAL(CronEd.PR.Setpoint[92])/10; runs INTERN ASSIGN CronEd.PR.Setpoint[92]:=(REAL_TO_WORD(CronEd.PR_TT*10))
rounded rectangle at (570,692)-(601,708): text "%.1f"; shows WORD_TO_REAL(CronEd.PR.Setpoint[93])/10; runs INTERN ASSIGN CronEd.PR.Setpoint[93]:=(REAL_TO_WORD(CronEd.PR_TT*10))
rounded rectangle at (570,707)-(601,723): text "%.1f"; shows WORD_TO_REAL(CronEd.PR.Setpoint[94])/10; runs INTERN ASSIGN CronEd.PR.Setpoint[94]:=(REAL_TO_WORD(CronEd.PR_TT*10))
rounded rectangle at (570,722)-(601,738): text "%.1f"; shows WORD_TO_REAL(CronEd.PR.Setpoint[95])/10; runs INTERN ASSIGN CronEd.PR.Setpoint[95]:=(REAL_TO_WORD(CronEd.PR_TT*10))
rounded rectangle at (570,737)-(601,753): text "%.1f"; shows WORD_TO_REAL(CronEd.PR.Setpoint[96])/10; runs INTERN ASSIGN CronEd.PR.Setpoint[96]:=(REAL_TO_WORD(CronEd.PR_TT*10))
rounded rectangle at (570,752)-(601,768): text "%.1f"; shows WORD_TO_REAL(CronEd.PR.Setpoint[97])/10; runs INTERN ASSIGN CronEd.PR.Setpoint[97]:=(REAL_TO_WORD(CronEd.PR_TT*10))
rounded rectangle at (570,767)-(601,783): text "%.1f"; shows WORD_TO_REAL(CronEd.PR.Setpoint[98])/10; runs INTERN ASSIGN CronEd.PR.Setpoint[98]:=(REAL_TO_WORD(CronEd.PR_TT*10))
rounded rectangle at (570,782)-(601,798): text "%.1f"; shows WORD_TO_REAL(CronEd.PR.Setpoint[99])/10; runs INTERN ASSIGN CronEd.PR.Setpoint[99]:=(REAL_TO_WORD(CronEd.PR_TT*10))
rounded rectangle at (570,796)-(601,812): text "%.1f"; shows WORD_TO_REAL(CronEd.PR.Setpoint[100])/10; runs INTERN ASSIGN CronEd.PR.Setpoint[100]:=(REAL_TO_WORD(CronEd.PR_TT*10))
rounded rectangle at (570,811)-(601,827): text "%.1f"; shows WORD_TO_REAL(CronEd.PR.Setpoint[101])/10; runs INTERN ASSIGN CronEd.PR.Setpoint[101]:=(REAL_TO_WORD(CronEd.PR_TT*10))
rounded rectangle at (570,826)-(601,842): text "%.1f"; shows WORD_TO_REAL(CronEd.PR.Setpoint[102])/10; runs INTERN ASSIGN CronEd.PR.Setpoint[102]:=(REAL_TO_WORD(CronEd.PR_TT*10))
rounded rectangle at (570,841)-(601,857): text "%.1f"; shows WORD_TO_REAL(CronEd.PR.Setpoint[103])/10; runs INTERN ASSIGN CronEd.PR.Setpoint[103]:=(REAL_TO_WORD(CronEd.PR_TT*10))
rounded rectangle at (570,855)-(601,871): text "%.1f"; shows WORD_TO_REAL(CronEd.PR.Setpoint[104])/10; runs INTERN ASSIGN CronEd.PR.Setpoint[104]:=(REAL_TO_WORD(CronEd.PR_TT*10))
rounded rectangle at (570,870)-(601,886): text "%.1f"; shows WORD_TO_REAL(CronEd.PR.Setpoint[105])/10; runs INTERN ASSIGN CronEd.PR.Setpoint[105]:=(REAL_TO_WORD(CronEd.PR_TT*10))
rounded rectangle at (570,885)-(601,901): text "%.1f"; shows WORD_TO_REAL(CronEd.PR.Setpoint[106])/10; runs INTERN ASSIGN CronEd.PR.Setpoint[106]:=(REAL_TO_WORD(CronEd.PR_TT*10))
rounded rectangle at (570,900)-(601,916): text "%.1f"; shows WORD_TO_REAL(CronEd.PR.Setpoint[107])/10; runs INTERN ASSIGN CronEd.PR.Setpoint[107]:=(REAL_TO_WORD(CronEd.PR_TT*10))
rounded rectangle at (570,914)-(601,930): text "%.1f"; shows WORD_TO_REAL(CronEd.PR.Setpoint[1068])/10; runs INTERN ASSIGN CronEd.PR.Setpoint[1068]:=(REAL_TO_WORD(CronEd.PR_TT*10))
rounded rectangle at (570,929)-(601,945): text "%.1f"; shows WORD_TO_REAL(CronEd.PR.Setpoint[1069])/10; runs INTERN ASSIGN CronEd.PR.Setpoint[1069]:=(REAL_TO_WORD(CronEd.PR_TT*10))
rounded rectangle at (570,944)-(601,960): text "%.1f"; shows WORD_TO_REAL(CronEd.PR.Setpoint[1070])/10; runs INTERN ASSIGN CronEd.PR.Setpoint[1070]:=(REAL_TO_WORD(CronEd.PR_TT*10))
rounded rectangle at (570,959)-(601,975): text "%.1f"; shows WORD_TO_REAL(CronEd.PR.Setpoint[1071])/10; runs INTERN ASSIGN CronEd.PR.Setpoint[1071]:=(REAL_TO_WORD(CronEd.PR_TT*10))
rounded rectangle at (570,973)-(601,989): text "%.1f"; shows WORD_TO_REAL(CronEd.PR.Setpoint[1072])/10; runs INTERN ASSIGN CronEd.PR.Setpoint[1072]:=(REAL_TO_WORD(CronEd.PR_TT*10))
rounded rectangle at (570,988)-(601,1004): text "%.1f"; shows WORD_TO_REAL(CronEd.PR.Setpoint[1073])/10; runs INTERN ASSIGN CronEd.PR.Setpoint[1073]:=(REAL_TO_WORD(CronEd.PR_TT*10))
rounded rectangle at (570,1003)-(601,1019): text "%.1f"; shows WORD_TO_REAL(CronEd.PR.Setpoint[1074])/10; runs INTERN ASSIGN CronEd.PR.Setpoint[1074]:=(REAL_TO_WORD(CronEd.PR_TT*10))
rounded rectangle at (570,1018)-(601,1034): text "%.1f"; shows WORD_TO_REAL(CronEd.PR.Setpoint[1075])/10; runs INTERN ASSIGN CronEd.PR.Setpoint[1075]:=(REAL_TO_WORD(CronEd.PR_TT*10))
rounded rectangle at (570,1033)-(601,1049): text "%.1f"; shows WORD_TO_REAL(CronEd.PR.Setpoint[1076])/10; runs INTERN ASSIGN CronEd.PR.Setpoint[1076]:=(REAL_TO_WORD(CronEd.PR_TT*10))
rounded rectangle at (570,1048)-(601,1064): text "%.1f"; shows WORD_TO_REAL(CronEd.PR.Setpoint[1077])/10; runs INTERN ASSIGN CronEd.PR.Setpoint[1077]:=(REAL_TO_WORD(CronEd.PR_TT*10))
rounded rectangle at (570,1063)-(601,1079): text "%.1f"; shows WORD_TO_REAL(CronEd.PR.Setpoint[1078])/10; runs INTERN ASSIGN CronEd.PR.Setpoint[1078]:=(REAL_TO_WORD(CronEd.PR_TT*10))
rounded rectangle at (570,1078)-(601,1094): text "%.1f"; shows WORD_TO_REAL(CronEd.PR.Setpoint[1079])/10; runs INTERN ASSIGN CronEd.PR.Setpoint[1079]:=(REAL_TO_WORD(CronEd.PR_TT*10))
2 more shapes without text or variables
*)
